// TIA Portal V17 program export: 1 tag tables, 0 data types, 2 data blocks, 8 code blocks (in call order from the OBs), 3 instance data blocks

VAR_GLOBAL   // PLC tag table "System"
   System_Byte AT %MB1 : Byte;
   FirstScan AT %M1.0 : Bool;
   DiagStatusUpdate AT %M1.1 : Bool;
   AlwaysTRUE AT %M1.2 : Bool;
   AlwaysFALSE AT %M1.3 : Bool;
   Clock_Byte AT %MB0 : Byte;
   Clock_10Hz AT %M0.0 : Bool;
   Clock_5Hz AT %M0.1 : Bool;
   "Clock_2.5Hz" AT %M0.2 : Bool;
   Clock_2Hz AT %M0.3 : Bool;
   "Clock_1.25Hz" AT %M0.4 : Bool;
   Clock_1Hz AT %M0.5 : Bool;
   "Clock_0.625Hz" AT %M0.6 : Bool;
   "Clock_0.5Hz" AT %M0.7 : Bool;
   Tag_1 AT %MD100 : DWord;
END_VAR

DATA_BLOCK "Modbus RTU buffer"   // DB11
{ S7_Optimized_Access := 'FALSE' }
VERSION : 0.1
// stored: AutoNumber false, DBAccessibleFromOPCUA true, IsOnlyStoredInLoadMemory false, IsWriteProtectedInAS false
   VAR
      "Operation data number_H" { ExternalAccessible := 'False'; ExternalVisible := 'False'; ExternalWritable := 'False'} : UInt;   // Modbus register 88
      "Operation data number_L" { ExternalAccessible := 'False'; ExternalVisible := 'False'; ExternalWritable := 'False'} : UInt;   // Modbus register 89
      "Operation type_H" { ExternalAccessible := 'False'; ExternalVisible := 'False'; ExternalWritable := 'False'} : UInt;   // Modbus register 90
      "Operation type_L" { ExternalAccessible := 'False'; ExternalVisible := 'False'; ExternalWritable := 'False'} : UInt;   // Modbus register 91
      Position_H { ExternalAccessible := 'False'; ExternalVisible := 'False'; ExternalWritable := 'False'} : UInt;   // Modbus register 92
      Position_L { ExternalAccessible := 'False'; ExternalVisible := 'False'; ExternalWritable := 'False'} : UInt;   // Modbus register 93
      Speed_H { ExternalAccessible := 'False'; ExternalVisible := 'False'; ExternalWritable := 'False'} : UInt;   // Modbus register 94
      Speed_L { ExternalAccessible := 'False'; ExternalVisible := 'False'; ExternalWritable := 'False'} : UInt;   // Modbus register 95
      "Starting_Changing rate_H" { ExternalAccessible := 'False'; ExternalVisible := 'False'; ExternalWritable := 'False'} : UInt;   // Modbus register 96
      "Starting_Changing rate_L" { ExternalAccessible := 'False'; ExternalVisible := 'False'; ExternalWritable := 'False'} : UInt;   // Modbus register 97
      "Stopping deceleration_H" { ExternalAccessible := 'False'; ExternalVisible := 'False'; ExternalWritable := 'False'} : UInt;   // Modbus register 98
      "Stopping deceleration_L" { ExternalAccessible := 'False'; ExternalVisible := 'False'; ExternalWritable := 'False'} : UInt;   // Modbus register 99
      "Operating current_H" { ExternalAccessible := 'False'; ExternalVisible := 'False'; ExternalWritable := 'False'} : UInt;   // Modbus register 100
      "Operating current_L" { ExternalAccessible := 'False'; ExternalVisible := 'False'; ExternalWritable := 'False'} : UInt;   // Modbus register 101
      "Operation trigger_H" { ExternalAccessible := 'False'; ExternalVisible := 'False'; ExternalWritable := 'False'} : UInt;   // Modbus register 102
      "Operation trigger_L" { ExternalAccessible := 'False'; ExternalVisible := 'False'; ExternalWritable := 'False'} : UInt;   // Modbus register 103
      "Forwarding destination_H" { ExternalAccessible := 'False'; ExternalVisible := 'False'; ExternalWritable := 'False'} : UInt;   // Modbus register 104
      "Forwarding destination_L" { ExternalAccessible := 'False'; ExternalVisible := 'False'; ExternalWritable := 'False'} : UInt;   // Modbus register 105
      "Alarm reset_H" { ExternalAccessible := 'False'; ExternalVisible := 'False'; ExternalWritable := 'False'} : UInt;   // Modbus register 384
      "Alarm reset_L" { ExternalAccessible := 'False'; ExternalVisible := 'False'; ExternalWritable := 'False'} : UInt;   // Modbus register 385
      "Clear Monitor alarm history_H" { ExternalAccessible := 'False'; ExternalVisible := 'False'; ExternalWritable := 'False'} : UInt;   // Modbus register 388
      "Clear Monitor alarm history_L" { ExternalAccessible := 'False'; ExternalVisible := 'False'; ExternalWritable := 'False'} : UInt;   // Modbus register 389
      "Clear comm history_H" { ExternalAccessible := 'False'; ExternalVisible := 'False'; ExternalWritable := 'False'} : UInt;   // Modbus register 392
      "Clear comm history_L" { ExternalAccessible := 'False'; ExternalVisible := 'False'; ExternalWritable := 'False'} : UInt;   // Modbus register 393
      "Monitor present alarm_H" { ExternalAccessible := 'False'; ExternalVisible := 'False'; ExternalWritable := 'False'} : UInt;   // Modbus register 128
      "Monitor present alarm_L" { ExternalAccessible := 'False'; ExternalVisible := 'False'; ExternalWritable := 'False'} : UInt;   // Modbus register 129
      "Monitor alarm history 1_H" { ExternalAccessible := 'False'; ExternalVisible := 'False'; ExternalWritable := 'False'} : UInt;   // Modbus register 130
      "Monitor alarm history 1_L" { ExternalAccessible := 'False'; ExternalVisible := 'False'; ExternalWritable := 'False'} : UInt;   // Modbus register 131
      "Monitor alarm history 2_H" { ExternalAccessible := 'False'; ExternalVisible := 'False'; ExternalWritable := 'False'} : UInt;   // Modbus register 132
      "Monitor alarm history 2_L" { ExternalAccessible := 'False'; ExternalVisible := 'False'; ExternalWritable := 'False'} : UInt;   // Modbus register 133
      "Monitor alarm history 3_H" { ExternalAccessible := 'False'; ExternalVisible := 'False'; ExternalWritable := 'False'} : UInt;   // Modbus register 134
      "Monitor alarm history 3_L" { ExternalAccessible := 'False'; ExternalVisible := 'False'; ExternalWritable := 'False'} : UInt;   // Modbus register 135
      "Monitor alarm history 4_H" { ExternalAccessible := 'False'; ExternalVisible := 'False'; ExternalWritable := 'False'} : UInt;   // Modbus register 136
      "Monitor alarm history 4_L" { ExternalAccessible := 'False'; ExternalVisible := 'False'; ExternalWritable := 'False'} : UInt;   // Modbus register 137
      "Monitor alarm history 5_H" { ExternalAccessible := 'False'; ExternalVisible := 'False'; ExternalWritable := 'False'} : UInt;   // Modbus register 138
      "Monitor alarm history 5_L" { ExternalAccessible := 'False'; ExternalVisible := 'False'; ExternalWritable := 'False'} : UInt;   // Modbus register 139
      "Monitor present communication error_H" { ExternalAccessible := 'False'; ExternalVisible := 'False'; ExternalWritable := 'False'} : UInt;   // Modbus register 172
      "Monitor present communication error_L" { ExternalAccessible := 'False'; ExternalVisible := 'False'; ExternalWritable := 'False'} : UInt;   // Modbus register 173
      "Monitor communication error history 1_H" { ExternalAccessible := 'False'; ExternalVisible := 'False'; ExternalWritable := 'False'} : UInt;   // Modbus register 174
      "Monitor communication error history 1_L" { ExternalAccessible := 'False'; ExternalVisible := 'False'; ExternalWritable := 'False'} : UInt;   // Modbus register 175
      "Monitor communication error history 2_H" { ExternalAccessible := 'False'; ExternalVisible := 'False'; ExternalWritable := 'False'} : UInt;   // Modbus register 176
      "Monitor communication error history 2_L" { ExternalAccessible := 'False'; ExternalVisible := 'False'; ExternalWritable := 'False'} : UInt;   // Modbus register 177
      "Monitor communication error history 3_H" { ExternalAccessible := 'False'; ExternalVisible := 'False'; ExternalWritable := 'False'} : UInt;   // Modbus register 178
      "Monitor communication error history 3_L" { ExternalAccessible := 'False'; ExternalVisible := 'False'; ExternalWritable := 'False'} : UInt;   // Modbus register 179
      "Monitor communication error history 4_H" { ExternalAccessible := 'False'; ExternalVisible := 'False'; ExternalWritable := 'False'} : UInt;   // Modbus register 180
      "Monitor communication error history 4_L" { ExternalAccessible := 'False'; ExternalVisible := 'False'; ExternalWritable := 'False'} : UInt;   // Modbus register 181
      "Monitor communication error history 5_H" { ExternalAccessible := 'False'; ExternalVisible := 'False'; ExternalWritable := 'False'} : UInt;   // Modbus register 182
      "Monitor communication error history 5_L" { ExternalAccessible := 'False'; ExternalVisible := 'False'; ExternalWritable := 'False'} : UInt;   // Modbus register 183
      "Monitor feedback position_H" { ExternalAccessible := 'False'; ExternalVisible := 'False'; ExternalWritable := 'False'} : UInt;   // Modbus register 204
      "Monitor feedback position_L" { ExternalAccessible := 'False'; ExternalVisible := 'False'; ExternalWritable := 'False'} : UInt;   // Modbus register 205
      "Monitor feedback speed r/min_H" { ExternalAccessible := 'False'; ExternalVisible := 'False'; ExternalWritable := 'False'} : UInt;   // Modbus register 206
      "Monitor feedback speed r/min_L" { ExternalAccessible := 'False'; ExternalVisible := 'False'; ExternalWritable := 'False'} : UInt;   // Modbus register 207
      "Monitor feedback speed Hz_H" { ExternalAccessible := 'False'; ExternalVisible := 'False'; ExternalWritable := 'False'} : UInt;   // Modbus register 208
      "Monitor feedback speed Hz_L" { ExternalAccessible := 'False'; ExternalVisible := 'False'; ExternalWritable := 'False'} : UInt;   // Modbus register 209
      "Monitor direct I/O_H" { ExternalAccessible := 'False'; ExternalVisible := 'False'; ExternalWritable := 'False'} : UInt;   // Modbus register 212
      "Monitor direct I/O_L" { ExternalAccessible := 'False'; ExternalVisible := 'False'; ExternalWritable := 'False'} : UInt;   // Modbus register 213
      "Monitor torque_H" { ExternalAccessible := 'False'; ExternalVisible := 'False'; ExternalWritable := 'False'} : UInt;   // Modbus register 214
      "Monitor torque_L" { ExternalAccessible := 'False'; ExternalVisible := 'False'; ExternalWritable := 'False'} : UInt;   // Modbus register 215
      "Monitor cumulative load_H" { ExternalAccessible := 'False'; ExternalVisible := 'False'; ExternalWritable := 'False'} : UInt;   // Modbus register 218
      "Monitor cumulative load_L" { ExternalAccessible := 'False'; ExternalVisible := 'False'; ExternalWritable := 'False'} : UInt;   // Modbus register 219
      "Monitor driver temperature_H" { ExternalAccessible := 'False'; ExternalVisible := 'False'; ExternalWritable := 'False'} : UInt;   // Modbus register 248
      "Monitor driver temperature_L" { ExternalAccessible := 'False'; ExternalVisible := 'False'; ExternalWritable := 'False'} : UInt;   // Modbus register 249
      "Monitor motor temperature_H" { ExternalAccessible := 'False'; ExternalVisible := 'False'; ExternalWritable := 'False'} : UInt;   // Modbus register 250
      "Monitor motor temperature_L" { ExternalAccessible := 'False'; ExternalVisible := 'False'; ExternalWritable := 'False'} : UInt;   // Modbus register 251
      "Monitor inverter voltage_H" { ExternalAccessible := 'False'; ExternalVisible := 'False'; ExternalWritable := 'False'} : UInt;   // Modbus register 326
      "Monitor inverter voltage_L" { ExternalAccessible := 'False'; ExternalVisible := 'False'; ExternalWritable := 'False'} : UInt;   // Modbus register 327
      "Monitor power supply voltage_H" { ExternalAccessible := 'False'; ExternalVisible := 'False'; ExternalWritable := 'False'} : UInt;   // Modbus register 328
      "Monitor power supply voltage_L" { ExternalAccessible := 'False'; ExternalVisible := 'False'; ExternalWritable := 'False'} : UInt;   // Modbus register 329
      "Monitor DIP SW_H" { ExternalAccessible := 'False'; ExternalVisible := 'False'; ExternalWritable := 'False'} : UInt;   // Modbus register 330
      "Monitor DIP SW_L" { ExternalAccessible := 'False'; ExternalVisible := 'False'; ExternalWritable := 'False'} : UInt;   // Modbus register 331
      "Monitor ROT SW0_H" { ExternalAccessible := 'False'; ExternalVisible := 'False'; ExternalWritable := 'False'} : UInt;   // Modbus register 332
      "Monitor ROT SW0_L" { ExternalAccessible := 'False'; ExternalVisible := 'False'; ExternalWritable := 'False'} : UInt;   // Modbus register 333
      "Monitor ROT SW1_H" { ExternalAccessible := 'False'; ExternalVisible := 'False'; ExternalWritable := 'False'} : UInt;   // Modbus register 334
      "Monitor ROT SW1_L" { ExternalAccessible := 'False'; ExternalVisible := 'False'; ExternalWritable := 'False'} : UInt;   // Modbus register 335
   END_VAR
BEGIN
END_DATA_BLOCK

DATA_BLOCK "Modbus RTU comm"   // DB10
{ S7_Optimized_Access := 'TRUE' }
VERSION : 0.1
// stored: AutoNumber false, DBAccessibleFromOPCUA true, IsOnlyStoredInLoadMemory false, IsRetainMemResEnabled false, IsWriteProtectedInAS false, MemoryReserve 100
   VAR
      "Setup Done" { ExternalAccessible := 'False'; ExternalVisible := 'False'; ExternalWritable := 'False'} : Bool;
      Sequencer : USInt;
      REQ { ExternalAccessible := 'False'; ExternalVisible := 'False'; ExternalWritable := 'False'} : Bool;
      BUSY : Bool;
      DONE : Bool;
      MB_ADDR { ExternalAccessible := 'False'; ExternalVisible := 'False'; ExternalWritable := 'False'} : Word;
      MODE { ExternalAccessible := 'False'; ExternalVisible := 'False'; ExternalWritable := 'False'} : USInt;
      "DATA ADDR" { ExternalAccessible := 'False'; ExternalVisible := 'False'; ExternalWritable := 'False'} : UDInt;
      DATA_LEN { ExternalAccessible := 'False'; ExternalVisible := 'False'; ExternalWritable := 'False'} : UInt;
      DATA_PTR : UInt;
   END_VAR
BEGIN
END_DATA_BLOCK

ORGANIZATION_BLOCK "Main"   // OB1, LAD, ProgramCycle
TITLE = "Main Program Sweep (Cycle)"
{ S7_Optimized_Access := 'TRUE' }
VERSION : 0.1
// stored: AutoNumber true, IsIECCheckEnabled false, SetENOAutomatically false
   VAR_INPUT
      Initial_Call : Bool;   // Initial call of this OB
      Remanence : Bool;   // =True, if remanent data are available
   END_VAR
BEGIN

REGION Network 1: Call Modbus RTU program blocks
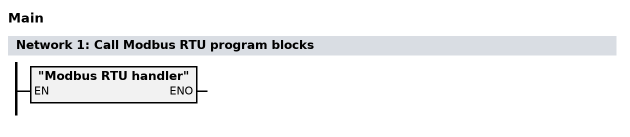
   RUNG wire#powerrail
      "Modbus RTU handler"()
   END_RUNG
   // the same network as SCL:
   "Modbus RTU handler"();
END_REGION
END_ORGANIZATION_BLOCK

FUNCTION "Modbus RTU handler" : Void   // FC10, LAD
TITLE = Modbus RTU handler
{ S7_Optimized_Access := 'TRUE' }
VERSION : 0.1
// This block updates R/W data from all the devices connected to the designated CM 1241 module.
// 
// Peripherals connected to this module:
// 
// -AZD-KD
// stored: AutoNumber false, IsIECCheckEnabled false, SetENOAutomatically false, UDAEnableTagReadback false
BEGIN

REGION Network 1: Modbus RTU module setup block
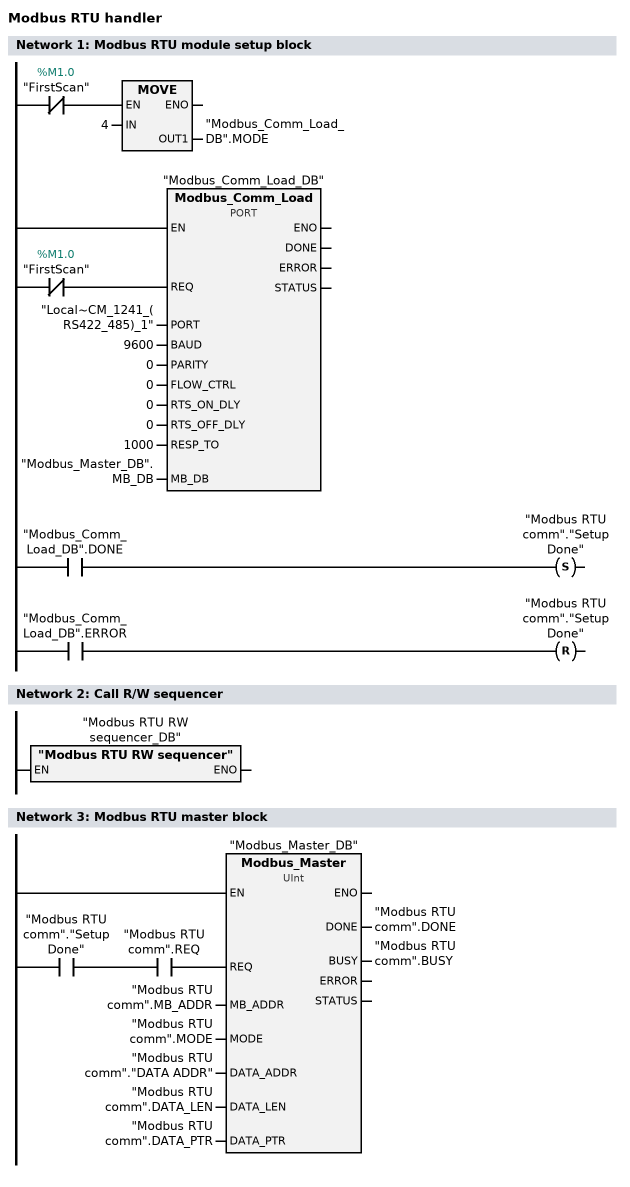
   RUNG wire#powerrail
      I_Contact( "FirstScan" )
      Move(in := 4, out1 => "Modbus_Comm_Load_DB".MODE)
   END_RUNG
   RUNG wire#powerrail
      { S7_Templates := "[card := 0, port_type := PORT, word_type := UInt, dint_type := UDInt, mbbase_type := P2P_MB_BASE]" } "Modbus_Comm_Load_DB".Modbus_Comm_Load(REQ := wire#w1, PORT := "Local~CM_1241_(RS422_485)_1", BAUD := 9600, PARITY := 0, FLOW_CTRL := 0, RTS_ON_DLY := 0, RTS_OFF_DLY := 0, RESP_TO := 1000, MB_DB := "Modbus_Master_DB".MB_DB, DONE =>, ERROR =>, STATUS =>)
   END_RUNG
   RUNG wire#powerrail
      I_Contact( "FirstScan" )
   END_RUNG wire#w1
   RUNG wire#powerrail
      Contact( "Modbus_Comm_Load_DB".DONE )
      S_Coil( "Modbus RTU comm"."Setup Done" )
   END_RUNG
   RUNG wire#powerrail
      Contact( "Modbus_Comm_Load_DB".ERROR )
      R_Coil( "Modbus RTU comm"."Setup Done" )
   END_RUNG
   // the same network as SCL:
   IF NOT "FirstScan" THEN "Modbus_Comm_Load_DB".MODE := 4; END_IF;
   "Modbus_Comm_Load_DB"(REQ := NOT "FirstScan",   // Modbus_Comm_Load
                         PORT := "Local~CM_1241_(RS422_485)_1",
                         BAUD := 9600,
                         PARITY := 0,
                         FLOW_CTRL := 0,
                         RTS_ON_DLY := 0,
                         RTS_OFF_DLY := 0,
                         RESP_TO := 1000,
                         MB_DB := "Modbus_Master_DB".MB_DB);
   IF "Modbus_Comm_Load_DB".DONE THEN "Modbus RTU comm"."Setup Done" := TRUE; END_IF;
   IF "Modbus_Comm_Load_DB".ERROR THEN "Modbus RTU comm"."Setup Done" := FALSE; END_IF;
END_REGION

REGION Network 2: Call R/W sequencer
   RUNG wire#powerrail
      "Modbus RTU RW sequencer_DB"()
   END_RUNG
   // the same network as SCL:
   "Modbus RTU RW sequencer_DB"();   // "Modbus RTU RW sequencer"
END_REGION

REGION Network 3: Modbus RTU master block
   RUNG wire#powerrail
      { S7_Templates := "[card := 0, word_type := UInt, dword_type := UDInt, byte_type := USInt, any_type := Variant]" } "Modbus_Master_DB".Modbus_Master(REQ := wire#w1, MB_ADDR := "Modbus RTU comm".MB_ADDR, MODE := "Modbus RTU comm".MODE, DATA_ADDR := "Modbus RTU comm"."DATA ADDR", DATA_LEN := "Modbus RTU comm".DATA_LEN, DATA_PTR := "Modbus RTU comm".DATA_PTR, DONE => "Modbus RTU comm".DONE, BUSY => "Modbus RTU comm".BUSY, ERROR =>, STATUS =>)
   END_RUNG
   RUNG wire#powerrail
      Contact( "Modbus RTU comm"."Setup Done" )
      Contact( "Modbus RTU comm".REQ )
   END_RUNG wire#w1
   // the same network as SCL:
   "Modbus_Master_DB"(REQ := "Modbus RTU comm"."Setup Done" AND "Modbus RTU comm".REQ,   // Modbus_Master
                      MB_ADDR := "Modbus RTU comm".MB_ADDR,
                      MODE := "Modbus RTU comm".MODE,
                      DATA_ADDR := "Modbus RTU comm"."DATA ADDR",
                      DATA_LEN := "Modbus RTU comm".DATA_LEN,
                      DATA_PTR := "Modbus RTU comm".DATA_PTR,
                      DONE => "Modbus RTU comm".DONE,
                      BUSY => "Modbus RTU comm".BUSY);
END_REGION
END_FUNCTION

FUNCTION_BLOCK "Modbus RTU RW sequencer"   // FB1, LAD
{ S7_Optimized_Access := 'TRUE' }
VERSION : 0.1
// stored: AutoNumber false, IsIECCheckEnabled false, IsRetainMemResEnabled false, MemoryReserve 100, SetENOAutomatically false, UDAEnableTagReadback false
   VAR
      "Operation data number" { S7_SetPoint := 'True'} : "Deconcatenate UDInt into two UInt";
      "Operation type" { S7_SetPoint := 'True'} : "Deconcatenate UDInt into two UInt";
      Position { S7_SetPoint := 'True'} : "Deconcatenate UDInt into two UInt";
      Speed { S7_SetPoint := 'True'} : "Deconcatenate UDInt into two UInt";
      "Starting changing rate" { S7_SetPoint := 'True'} : "Deconcatenate UDInt into two UInt";
      "Stopping deceleration" { S7_SetPoint := 'True'} : "Deconcatenate UDInt into two UInt";
      "Operating current" { S7_SetPoint := 'True'} : "Deconcatenate UDInt into two UInt";
      "Operation trigger" { S7_SetPoint := 'True'} : "Deconcatenate UDInt into two UInt";
      "Forwarding destination" { S7_SetPoint := 'True'} : "Deconcatenate UDInt into two UInt";
      "Alarm reset" { S7_SetPoint := 'True'} : "Deconcatenate UDInt into two UInt";
      "Clear alarm history" { S7_SetPoint := 'True'} : "Deconcatenate UDInt into two UInt";
      "Clear comm history" { S7_SetPoint := 'True'} : "Deconcatenate UDInt into two UInt";
      "Clear monitor alarm history" { S7_SetPoint := 'True'} : "Deconcatenate UDInt into two UInt";
      "Clear comm history_1" { S7_SetPoint := 'True'} : "Deconcatenate UDInt into two UInt";
      "Monitor present alarm" { S7_SetPoint := 'True'} : "Concatenate two UInt into one UDInt";
      "Monitor alarm history 1" { S7_SetPoint := 'True'} : "Concatenate two UInt into one UDInt";
      "Monitor alarm history 2" { S7_SetPoint := 'True'} : "Concatenate two UInt into one UDInt";
      "Monitor alarm history 3" { S7_SetPoint := 'True'} : "Concatenate two UInt into one UDInt";
      "Monitor alarm history 4" { S7_SetPoint := 'True'} : "Concatenate two UInt into one UDInt";
      "Monitor alarm history 5" { S7_SetPoint := 'True'} : "Concatenate two UInt into one UDInt";
      "Monitor present communication error" { S7_SetPoint := 'True'} : "Concatenate two UInt into one UDInt";
      "Monitor communication error history 1" { S7_SetPoint := 'True'} : "Concatenate two UInt into one UDInt";
      "Monitor communication error history 2" { S7_SetPoint := 'True'} : "Concatenate two UInt into one UDInt";
      "Monitor communication error history 3" { S7_SetPoint := 'True'} : "Concatenate two UInt into one UDInt";
      "Monitor communication error history 4" { S7_SetPoint := 'True'} : "Concatenate two UInt into one UDInt";
      "Monitor communication error history 5" { S7_SetPoint := 'True'} : "Concatenate two UInt into one UDInt";
      "Monitor feedback position" { S7_SetPoint := 'True'} : "Concatenate two UInt into one UDInt";
      "Monitor feedback speed r/min" { S7_SetPoint := 'True'} : "Concatenate two UInt into one UDInt";
      "Monitor feedback speed Hz" { S7_SetPoint := 'True'} : "Concatenate two UInt into one UDInt";
      "Monitor direct I/O" { S7_SetPoint := 'True'} : "Concatenate two UInt into one UDInt";
      "Monitor torque" { S7_SetPoint := 'True'} : "Concatenate two UInt into one UDInt";
      "Monitor cumulative load" { S7_SetPoint := 'True'} : "Concatenate two UInt into one UDInt";
      "Monitor driver temperature" { S7_SetPoint := 'True'} : "Concatenate two UInt into one UDInt";
      "Monitor motor temperature" { S7_SetPoint := 'True'} : "Concatenate two UInt into one UDInt";
      "Monitor inverter voltage" { S7_SetPoint := 'True'} : "Concatenate two UInt into one UDInt";
      "Monitor power supply voltage" { S7_SetPoint := 'True'} : "Concatenate two UInt into one UDInt";
      "Monitor DIP SW" { S7_SetPoint := 'True'} : "Concatenate two UInt into one UDInt";
      "Monitor ROT SW0" { S7_SetPoint := 'True'} : "Concatenate two UInt into one UDInt";
      "Monitor ROT SW1" { S7_SetPoint := 'True'} : "Concatenate two UInt into one UDInt";
   END_VAR
   VAR_TEMP   // added for the SCL form of the ladder/FBD networks
      _w1 : Bool;
   END_VAR
BEGIN

REGION Network 1: Deconcatenate data for writing it into modbus holding registers
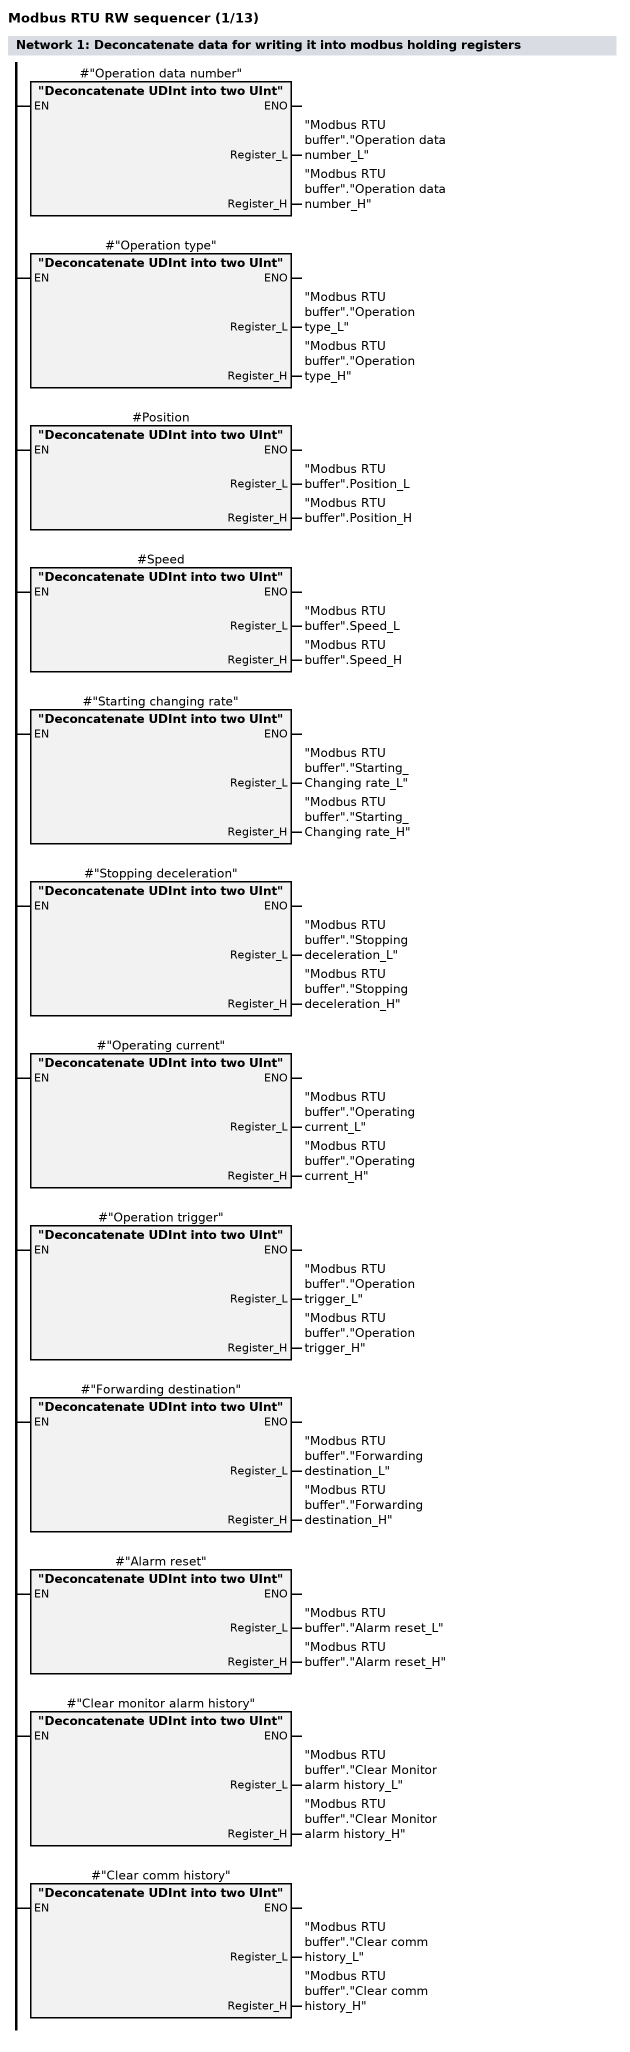
   RUNG wire#powerrail
      #"Operation data number"(Register_L => "Modbus RTU buffer"."Operation data number_L", Register_H => "Modbus RTU buffer"."Operation data number_H")
   END_RUNG
   RUNG wire#powerrail
      #"Operation type"(Register_L => "Modbus RTU buffer"."Operation type_L", Register_H => "Modbus RTU buffer"."Operation type_H")
   END_RUNG
   RUNG wire#powerrail
      #Position(Register_L => "Modbus RTU buffer".Position_L, Register_H => "Modbus RTU buffer".Position_H)
   END_RUNG
   RUNG wire#powerrail
      #Speed(Register_L => "Modbus RTU buffer".Speed_L, Register_H => "Modbus RTU buffer".Speed_H)
   END_RUNG
   RUNG wire#powerrail
      #"Starting changing rate"(Register_L => "Modbus RTU buffer"."Starting_Changing rate_L", Register_H => "Modbus RTU buffer"."Starting_Changing rate_H")
   END_RUNG
   RUNG wire#powerrail
      #"Stopping deceleration"(Register_L => "Modbus RTU buffer"."Stopping deceleration_L", Register_H => "Modbus RTU buffer"."Stopping deceleration_H")
   END_RUNG
   RUNG wire#powerrail
      #"Operating current"(Register_L => "Modbus RTU buffer"."Operating current_L", Register_H => "Modbus RTU buffer"."Operating current_H")
   END_RUNG
   RUNG wire#powerrail
      #"Operation trigger"(Register_L => "Modbus RTU buffer"."Operation trigger_L", Register_H => "Modbus RTU buffer"."Operation trigger_H")
   END_RUNG
   RUNG wire#powerrail
      #"Forwarding destination"(Register_L => "Modbus RTU buffer"."Forwarding destination_L", Register_H => "Modbus RTU buffer"."Forwarding destination_H")
   END_RUNG
   RUNG wire#powerrail
      #"Alarm reset"(Register_L => "Modbus RTU buffer"."Alarm reset_L", Register_H => "Modbus RTU buffer"."Alarm reset_H")
   END_RUNG
   RUNG wire#powerrail
      #"Clear monitor alarm history"(Register_L => "Modbus RTU buffer"."Clear Monitor alarm history_L", Register_H => "Modbus RTU buffer"."Clear Monitor alarm history_H")
   END_RUNG
   RUNG wire#powerrail
      #"Clear comm history"(Register_L => "Modbus RTU buffer"."Clear comm history_L", Register_H => "Modbus RTU buffer"."Clear comm history_H")
   END_RUNG
   // the same network as SCL:
   #"Operation data number"(Register_L => "Modbus RTU buffer"."Operation data number_L",   // "Deconcatenate UDInt into two UInt"
                           Register_H => "Modbus RTU buffer"."Operation data number_H");
   #"Operation type"(Register_L => "Modbus RTU buffer"."Operation type_L",   // "Deconcatenate UDInt into two UInt"
                     Register_H => "Modbus RTU buffer"."Operation type_H");
   #Position(Register_L => "Modbus RTU buffer".Position_L, Register_H => "Modbus RTU buffer".Position_H);   // "Deconcatenate UDInt into two UInt"
   #Speed(Register_L => "Modbus RTU buffer".Speed_L, Register_H => "Modbus RTU buffer".Speed_H);   // "Deconcatenate UDInt into two UInt"
   #"Starting changing rate"(Register_L => "Modbus RTU buffer"."Starting_Changing rate_L",   // "Deconcatenate UDInt into two UInt"
                           Register_H => "Modbus RTU buffer"."Starting_Changing rate_H");
   #"Stopping deceleration"(Register_L => "Modbus RTU buffer"."Stopping deceleration_L",   // "Deconcatenate UDInt into two UInt"
                           Register_H => "Modbus RTU buffer"."Stopping deceleration_H");
   #"Operating current"(Register_L => "Modbus RTU buffer"."Operating current_L",   // "Deconcatenate UDInt into two UInt"
                        Register_H => "Modbus RTU buffer"."Operating current_H");
   #"Operation trigger"(Register_L => "Modbus RTU buffer"."Operation trigger_L",   // "Deconcatenate UDInt into two UInt"
                        Register_H => "Modbus RTU buffer"."Operation trigger_H");
   #"Forwarding destination"(Register_L => "Modbus RTU buffer"."Forwarding destination_L",   // "Deconcatenate UDInt into two UInt"
                           Register_H => "Modbus RTU buffer"."Forwarding destination_H");
   #"Alarm reset"(Register_L => "Modbus RTU buffer"."Alarm reset_L",   // "Deconcatenate UDInt into two UInt"
                  Register_H => "Modbus RTU buffer"."Alarm reset_H");
   #"Clear monitor alarm history"(Register_L => "Modbus RTU buffer"."Clear Monitor alarm history_L",   // "Deconcatenate UDInt into two UInt"
                           Register_H => "Modbus RTU buffer"."Clear Monitor alarm history_H");
   #"Clear comm history"(Register_L => "Modbus RTU buffer"."Clear comm history_L",   // "Deconcatenate UDInt into two UInt"
                         Register_H => "Modbus RTU buffer"."Clear comm history_H");
END_REGION

REGION Network 2: Data writing/reading step 0: Write data from address 88 to address 105
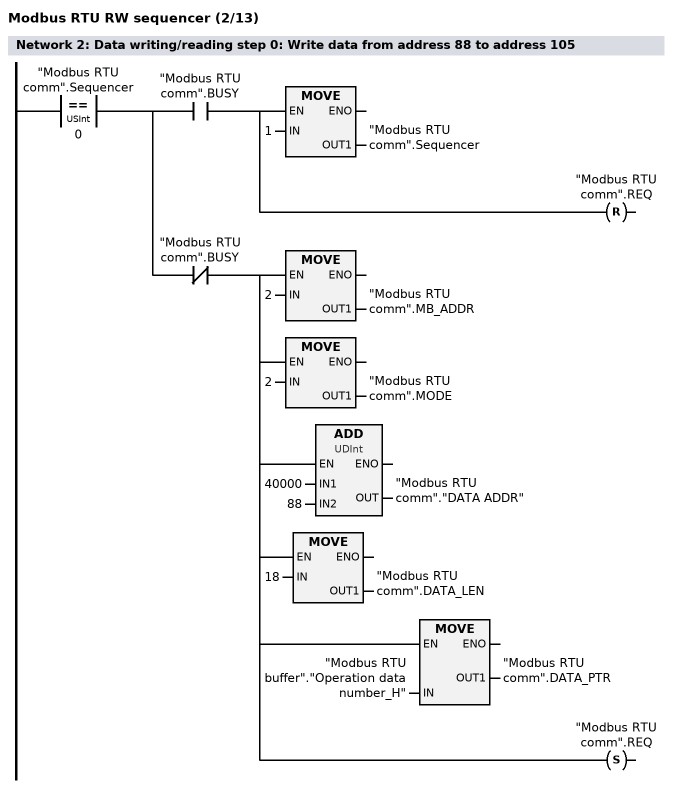
   RUNG wire#powerrail
      { S7_Templates := "SrcType := USInt" } EQ_Contact(in1 := "Modbus RTU comm".Sequencer, in2 := 0)
      wire#w1
      Contact( "Modbus RTU comm".BUSY )
      wire#w2
      Move(in := 1, out1 => "Modbus RTU comm".Sequencer)
   END_RUNG
   RUNG wire#w2
      R_Coil( "Modbus RTU comm".REQ )
   END_RUNG
   RUNG wire#w1
      I_Contact( "Modbus RTU comm".BUSY )
      wire#w3
      Move(in := 2, out1 => "Modbus RTU comm".MB_ADDR)
   END_RUNG
   RUNG wire#w3
      Move(in := 2, out1 => "Modbus RTU comm".MODE)
   END_RUNG
   RUNG wire#w3
      { S7_Templates := "SrcType := UDInt" } Add(in1 := 40000, in2 := 88, out => "Modbus RTU comm"."DATA ADDR")
   END_RUNG
   RUNG wire#w3
      Move(in := 18, out1 => "Modbus RTU comm".DATA_LEN)
   END_RUNG
   RUNG wire#w3
      Move(in := "Modbus RTU buffer"."Operation data number_H", out1 => "Modbus RTU comm".DATA_PTR)
   END_RUNG
   RUNG wire#w3
      S_Coil( "Modbus RTU comm".REQ )
   END_RUNG
   // the same network as SCL:
   #_w1 := "Modbus RTU comm".Sequencer = 0;
   IF #_w1 AND "Modbus RTU comm".BUSY THEN
       "Modbus RTU comm".Sequencer := 1;
       "Modbus RTU comm".REQ := FALSE;
   END_IF;
   IF #_w1 AND NOT "Modbus RTU comm".BUSY THEN
       "Modbus RTU comm".MB_ADDR := 2;
       "Modbus RTU comm".MODE := 2;
       "Modbus RTU comm"."DATA ADDR" := 40000 + 88;
       "Modbus RTU comm".DATA_LEN := 18;
       "Modbus RTU comm".DATA_PTR := "Modbus RTU buffer"."Operation data number_H";
       "Modbus RTU comm".REQ := TRUE;
   END_IF;
END_REGION

REGION Network 3: Data writing/reading step 1: Write data from address 384 to address 385
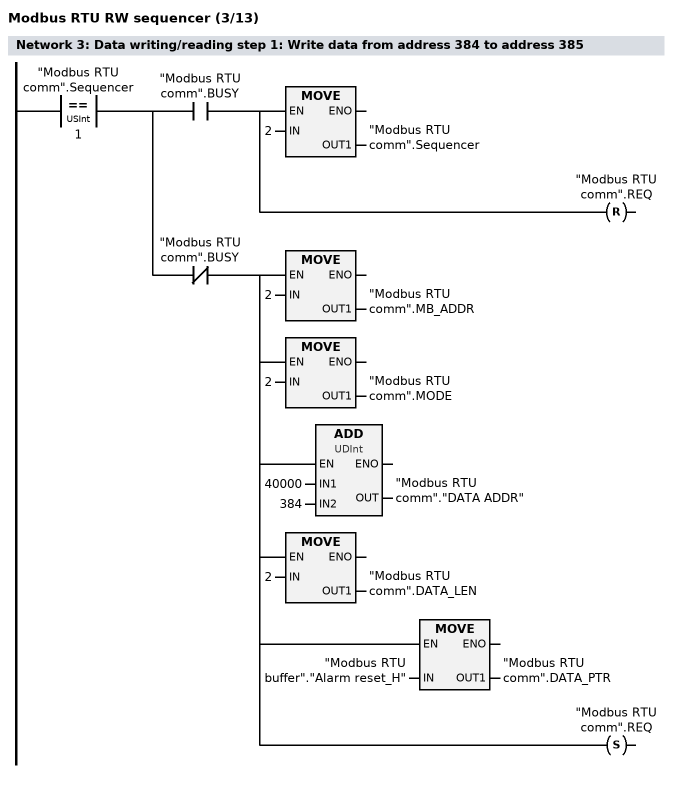
   RUNG wire#powerrail
      { S7_Templates := "SrcType := USInt" } EQ_Contact(in1 := "Modbus RTU comm".Sequencer, in2 := 1)
      wire#w1
      Contact( "Modbus RTU comm".BUSY )
      wire#w2
      Move(in := 2, out1 => "Modbus RTU comm".Sequencer)
   END_RUNG
   RUNG wire#w2
      R_Coil( "Modbus RTU comm".REQ )
   END_RUNG
   RUNG wire#w1
      I_Contact( "Modbus RTU comm".BUSY )
      wire#w3
      Move(in := 2, out1 => "Modbus RTU comm".MB_ADDR)
   END_RUNG
   RUNG wire#w3
      Move(in := 2, out1 => "Modbus RTU comm".MODE)
   END_RUNG
   RUNG wire#w3
      { S7_Templates := "SrcType := UDInt" } Add(in1 := 40000, in2 := 384, out => "Modbus RTU comm"."DATA ADDR")
   END_RUNG
   RUNG wire#w3
      Move(in := 2, out1 => "Modbus RTU comm".DATA_LEN)
   END_RUNG
   RUNG wire#w3
      Move(in := "Modbus RTU buffer"."Alarm reset_H", out1 => "Modbus RTU comm".DATA_PTR)
   END_RUNG
   RUNG wire#w3
      S_Coil( "Modbus RTU comm".REQ )
   END_RUNG
   // the same network as SCL:
   #_w1 := "Modbus RTU comm".Sequencer = 1;
   IF #_w1 AND "Modbus RTU comm".BUSY THEN
       "Modbus RTU comm".Sequencer := 2;
       "Modbus RTU comm".REQ := FALSE;
   END_IF;
   IF #_w1 AND NOT "Modbus RTU comm".BUSY THEN
       "Modbus RTU comm".MB_ADDR := 2;
       "Modbus RTU comm".MODE := 2;
       "Modbus RTU comm"."DATA ADDR" := 40000 + 384;
       "Modbus RTU comm".DATA_LEN := 2;
       "Modbus RTU comm".DATA_PTR := "Modbus RTU buffer"."Alarm reset_H";
       "Modbus RTU comm".REQ := TRUE;
   END_IF;
END_REGION

REGION Network 4: Data writing/reading step 2: Write data from address 388 to address 389
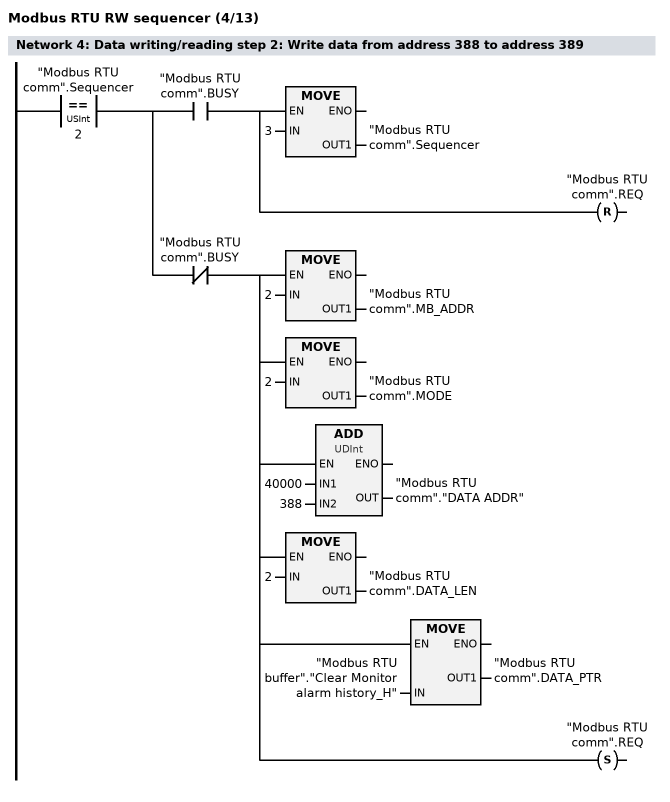
   RUNG wire#powerrail
      { S7_Templates := "SrcType := USInt" } EQ_Contact(in1 := "Modbus RTU comm".Sequencer, in2 := 2)
      wire#w1
      Contact( "Modbus RTU comm".BUSY )
      wire#w2
      Move(in := 3, out1 => "Modbus RTU comm".Sequencer)
   END_RUNG
   RUNG wire#w2
      R_Coil( "Modbus RTU comm".REQ )
   END_RUNG
   RUNG wire#w1
      I_Contact( "Modbus RTU comm".BUSY )
      wire#w3
      Move(in := 2, out1 => "Modbus RTU comm".MB_ADDR)
   END_RUNG
   RUNG wire#w3
      Move(in := 2, out1 => "Modbus RTU comm".MODE)
   END_RUNG
   RUNG wire#w3
      { S7_Templates := "SrcType := UDInt" } Add(in1 := 40000, in2 := 388, out => "Modbus RTU comm"."DATA ADDR")
   END_RUNG
   RUNG wire#w3
      Move(in := 2, out1 => "Modbus RTU comm".DATA_LEN)
   END_RUNG
   RUNG wire#w3
      Move(in := "Modbus RTU buffer"."Clear Monitor alarm history_H", out1 => "Modbus RTU comm".DATA_PTR)
   END_RUNG
   RUNG wire#w3
      S_Coil( "Modbus RTU comm".REQ )
   END_RUNG
   // the same network as SCL:
   #_w1 := "Modbus RTU comm".Sequencer = 2;
   IF #_w1 AND "Modbus RTU comm".BUSY THEN
       "Modbus RTU comm".Sequencer := 3;
       "Modbus RTU comm".REQ := FALSE;
   END_IF;
   IF #_w1 AND NOT "Modbus RTU comm".BUSY THEN
       "Modbus RTU comm".MB_ADDR := 2;
       "Modbus RTU comm".MODE := 2;
       "Modbus RTU comm"."DATA ADDR" := 40000 + 388;
       "Modbus RTU comm".DATA_LEN := 2;
       "Modbus RTU comm".DATA_PTR := "Modbus RTU buffer"."Clear Monitor alarm history_H";
       "Modbus RTU comm".REQ := TRUE;
   END_IF;
END_REGION

REGION Network 5: Data writing/reading step 3: Write data from address 392 to address 393
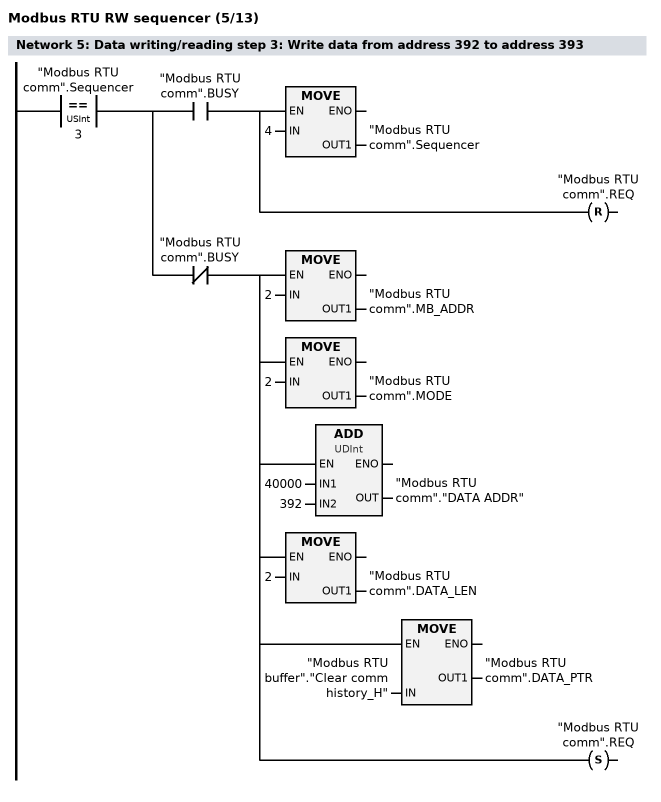
   RUNG wire#powerrail
      { S7_Templates := "SrcType := USInt" } EQ_Contact(in1 := "Modbus RTU comm".Sequencer, in2 := 3)
      wire#w1
      Contact( "Modbus RTU comm".BUSY )
      wire#w2
      Move(in := 4, out1 => "Modbus RTU comm".Sequencer)
   END_RUNG
   RUNG wire#w2
      R_Coil( "Modbus RTU comm".REQ )
   END_RUNG
   RUNG wire#w1
      I_Contact( "Modbus RTU comm".BUSY )
      wire#w3
      Move(in := 2, out1 => "Modbus RTU comm".MB_ADDR)
   END_RUNG
   RUNG wire#w3
      Move(in := 2, out1 => "Modbus RTU comm".MODE)
   END_RUNG
   RUNG wire#w3
      { S7_Templates := "SrcType := UDInt" } Add(in1 := 40000, in2 := 392, out => "Modbus RTU comm"."DATA ADDR")
   END_RUNG
   RUNG wire#w3
      Move(in := 2, out1 => "Modbus RTU comm".DATA_LEN)
   END_RUNG
   RUNG wire#w3
      Move(in := "Modbus RTU buffer"."Clear comm history_H", out1 => "Modbus RTU comm".DATA_PTR)
   END_RUNG
   RUNG wire#w3
      S_Coil( "Modbus RTU comm".REQ )
   END_RUNG
   // the same network as SCL:
   #_w1 := "Modbus RTU comm".Sequencer = 3;
   IF #_w1 AND "Modbus RTU comm".BUSY THEN
       "Modbus RTU comm".Sequencer := 4;
       "Modbus RTU comm".REQ := FALSE;
   END_IF;
   IF #_w1 AND NOT "Modbus RTU comm".BUSY THEN
       "Modbus RTU comm".MB_ADDR := 2;
       "Modbus RTU comm".MODE := 2;
       "Modbus RTU comm"."DATA ADDR" := 40000 + 392;
       "Modbus RTU comm".DATA_LEN := 2;
       "Modbus RTU comm".DATA_PTR := "Modbus RTU buffer"."Clear comm history_H";
       "Modbus RTU comm".REQ := TRUE;
   END_IF;
END_REGION

REGION Network 6: Data writing/reading step 4: Read data from address 128 to address 139
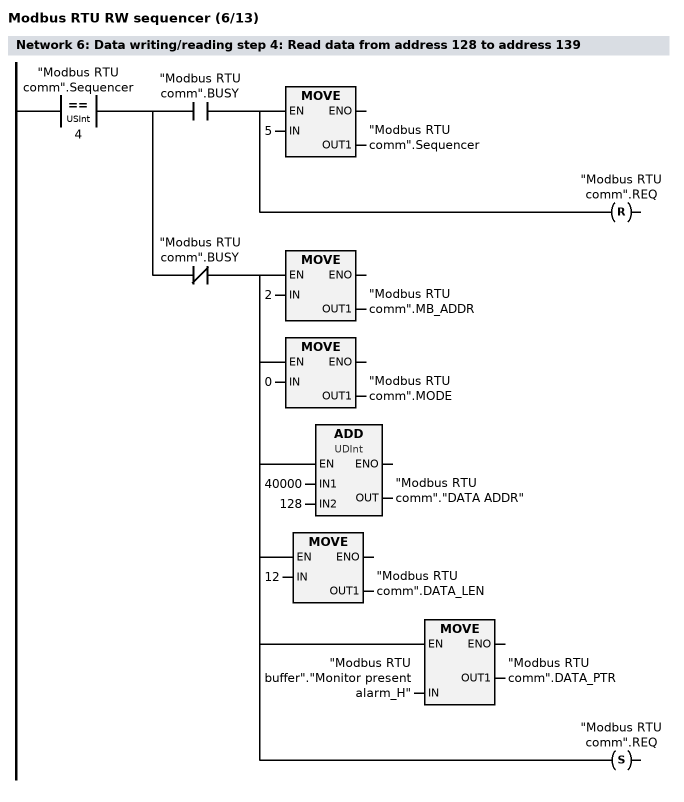
   RUNG wire#powerrail
      { S7_Templates := "SrcType := USInt" } EQ_Contact(in1 := "Modbus RTU comm".Sequencer, in2 := 4)
      wire#w1
      Contact( "Modbus RTU comm".BUSY )
      wire#w2
      Move(in := 5, out1 => "Modbus RTU comm".Sequencer)
   END_RUNG
   RUNG wire#w2
      R_Coil( "Modbus RTU comm".REQ )
   END_RUNG
   RUNG wire#w1
      I_Contact( "Modbus RTU comm".BUSY )
      wire#w3
      Move(in := 2, out1 => "Modbus RTU comm".MB_ADDR)
   END_RUNG
   RUNG wire#w3
      Move(in := 0, out1 => "Modbus RTU comm".MODE)
   END_RUNG
   RUNG wire#w3
      { S7_Templates := "SrcType := UDInt" } Add(in1 := 40000, in2 := 128, out => "Modbus RTU comm"."DATA ADDR")
   END_RUNG
   RUNG wire#w3
      Move(in := 12, out1 => "Modbus RTU comm".DATA_LEN)
   END_RUNG
   RUNG wire#w3
      Move(in := "Modbus RTU buffer"."Monitor present alarm_H", out1 => "Modbus RTU comm".DATA_PTR)
   END_RUNG
   RUNG wire#w3
      S_Coil( "Modbus RTU comm".REQ )
   END_RUNG
   // the same network as SCL:
   #_w1 := "Modbus RTU comm".Sequencer = 4;
   IF #_w1 AND "Modbus RTU comm".BUSY THEN
       "Modbus RTU comm".Sequencer := 5;
       "Modbus RTU comm".REQ := FALSE;
   END_IF;
   IF #_w1 AND NOT "Modbus RTU comm".BUSY THEN
       "Modbus RTU comm".MB_ADDR := 2;
       "Modbus RTU comm".MODE := 0;
       "Modbus RTU comm"."DATA ADDR" := 40000 + 128;
       "Modbus RTU comm".DATA_LEN := 12;
       "Modbus RTU comm".DATA_PTR := "Modbus RTU buffer"."Monitor present alarm_H";
       "Modbus RTU comm".REQ := TRUE;
   END_IF;
END_REGION

REGION Network 7: Data writing/reading step 5: Read data from address 172 to address 183
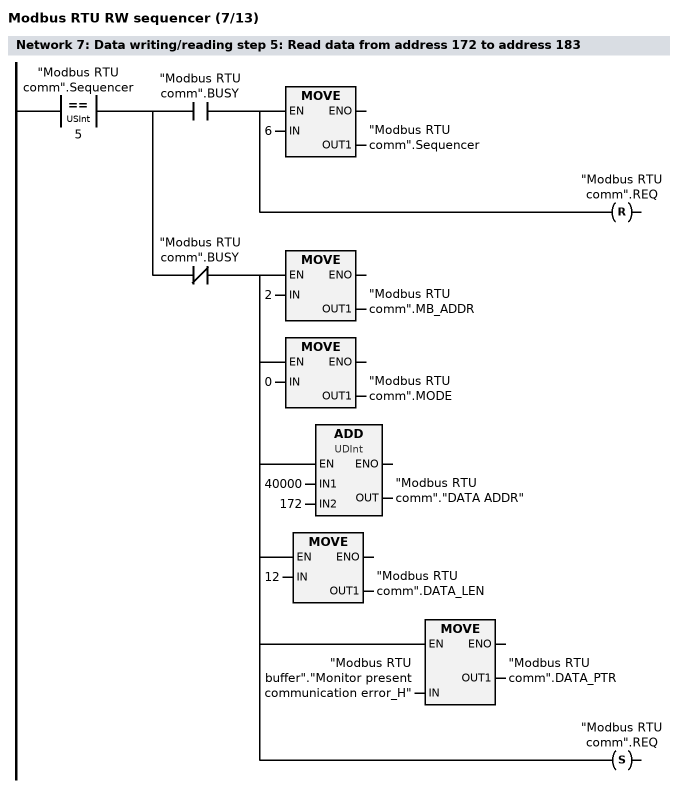
   RUNG wire#powerrail
      { S7_Templates := "SrcType := USInt" } EQ_Contact(in1 := "Modbus RTU comm".Sequencer, in2 := 5)
      wire#w1
      Contact( "Modbus RTU comm".BUSY )
      wire#w2
      Move(in := 6, out1 => "Modbus RTU comm".Sequencer)
   END_RUNG
   RUNG wire#w2
      R_Coil( "Modbus RTU comm".REQ )
   END_RUNG
   RUNG wire#w1
      I_Contact( "Modbus RTU comm".BUSY )
      wire#w3
      Move(in := 2, out1 => "Modbus RTU comm".MB_ADDR)
   END_RUNG
   RUNG wire#w3
      Move(in := 0, out1 => "Modbus RTU comm".MODE)
   END_RUNG
   RUNG wire#w3
      { S7_Templates := "SrcType := UDInt" } Add(in1 := 40000, in2 := 172, out => "Modbus RTU comm"."DATA ADDR")
   END_RUNG
   RUNG wire#w3
      Move(in := 12, out1 => "Modbus RTU comm".DATA_LEN)
   END_RUNG
   RUNG wire#w3
      Move(in := "Modbus RTU buffer"."Monitor present communication error_H", out1 => "Modbus RTU comm".DATA_PTR)
   END_RUNG
   RUNG wire#w3
      S_Coil( "Modbus RTU comm".REQ )
   END_RUNG
   // the same network as SCL:
   #_w1 := "Modbus RTU comm".Sequencer = 5;
   IF #_w1 AND "Modbus RTU comm".BUSY THEN
       "Modbus RTU comm".Sequencer := 6;
       "Modbus RTU comm".REQ := FALSE;
   END_IF;
   IF #_w1 AND NOT "Modbus RTU comm".BUSY THEN
       "Modbus RTU comm".MB_ADDR := 2;
       "Modbus RTU comm".MODE := 0;
       "Modbus RTU comm"."DATA ADDR" := 40000 + 172;
       "Modbus RTU comm".DATA_LEN := 12;
       "Modbus RTU comm".DATA_PTR := "Modbus RTU buffer"."Monitor present communication error_H";
       "Modbus RTU comm".REQ := TRUE;
   END_IF;
END_REGION

REGION Network 8: Data writing/reading step 6: Read data from address 204 to address 209
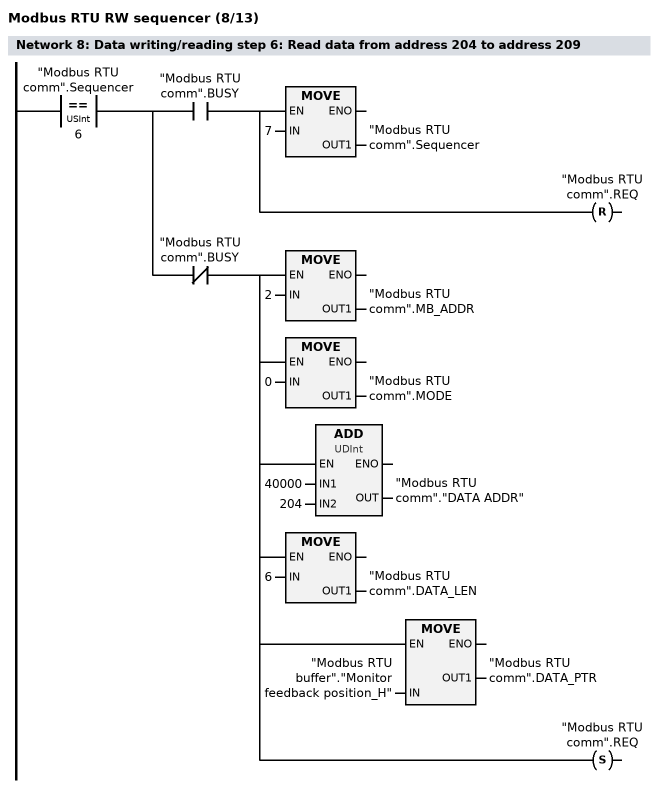
   RUNG wire#powerrail
      { S7_Templates := "SrcType := USInt" } EQ_Contact(in1 := "Modbus RTU comm".Sequencer, in2 := 6)
      wire#w1
      Contact( "Modbus RTU comm".BUSY )
      wire#w2
      Move(in := 7, out1 => "Modbus RTU comm".Sequencer)
   END_RUNG
   RUNG wire#w2
      R_Coil( "Modbus RTU comm".REQ )
   END_RUNG
   RUNG wire#w1
      I_Contact( "Modbus RTU comm".BUSY )
      wire#w3
      Move(in := 2, out1 => "Modbus RTU comm".MB_ADDR)
   END_RUNG
   RUNG wire#w3
      Move(in := 0, out1 => "Modbus RTU comm".MODE)
   END_RUNG
   RUNG wire#w3
      { S7_Templates := "SrcType := UDInt" } Add(in1 := 40000, in2 := 204, out => "Modbus RTU comm"."DATA ADDR")
   END_RUNG
   RUNG wire#w3
      Move(in := 6, out1 => "Modbus RTU comm".DATA_LEN)
   END_RUNG
   RUNG wire#w3
      Move(in := "Modbus RTU buffer"."Monitor feedback position_H", out1 => "Modbus RTU comm".DATA_PTR)
   END_RUNG
   RUNG wire#w3
      S_Coil( "Modbus RTU comm".REQ )
   END_RUNG
   // the same network as SCL:
   #_w1 := "Modbus RTU comm".Sequencer = 6;
   IF #_w1 AND "Modbus RTU comm".BUSY THEN
       "Modbus RTU comm".Sequencer := 7;
       "Modbus RTU comm".REQ := FALSE;
   END_IF;
   IF #_w1 AND NOT "Modbus RTU comm".BUSY THEN
       "Modbus RTU comm".MB_ADDR := 2;
       "Modbus RTU comm".MODE := 0;
       "Modbus RTU comm"."DATA ADDR" := 40000 + 204;
       "Modbus RTU comm".DATA_LEN := 6;
       "Modbus RTU comm".DATA_PTR := "Modbus RTU buffer"."Monitor feedback position_H";
       "Modbus RTU comm".REQ := TRUE;
   END_IF;
END_REGION

REGION Network 9: Data writing/reading step 7: Read data from address 212 to address 215
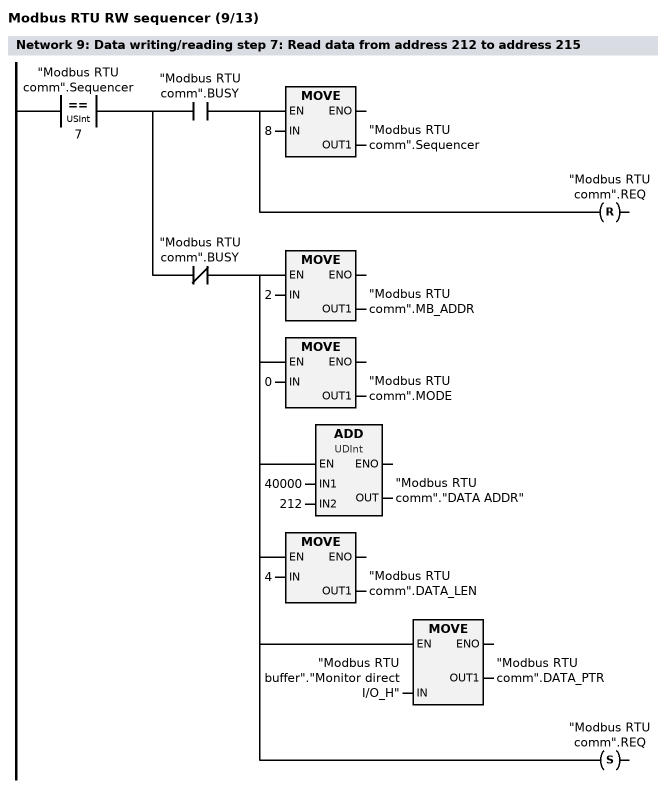
   RUNG wire#powerrail
      { S7_Templates := "SrcType := USInt" } EQ_Contact(in1 := "Modbus RTU comm".Sequencer, in2 := 7)
      wire#w1
      Contact( "Modbus RTU comm".BUSY )
      wire#w2
      Move(in := 8, out1 => "Modbus RTU comm".Sequencer)
   END_RUNG
   RUNG wire#w2
      R_Coil( "Modbus RTU comm".REQ )
   END_RUNG
   RUNG wire#w1
      I_Contact( "Modbus RTU comm".BUSY )
      wire#w3
      Move(in := 2, out1 => "Modbus RTU comm".MB_ADDR)
   END_RUNG
   RUNG wire#w3
      Move(in := 0, out1 => "Modbus RTU comm".MODE)
   END_RUNG
   RUNG wire#w3
      { S7_Templates := "SrcType := UDInt" } Add(in1 := 40000, in2 := 212, out => "Modbus RTU comm"."DATA ADDR")
   END_RUNG
   RUNG wire#w3
      Move(in := 4, out1 => "Modbus RTU comm".DATA_LEN)
   END_RUNG
   RUNG wire#w3
      Move(in := "Modbus RTU buffer"."Monitor direct I/O_H", out1 => "Modbus RTU comm".DATA_PTR)
   END_RUNG
   RUNG wire#w3
      S_Coil( "Modbus RTU comm".REQ )
   END_RUNG
   // the same network as SCL:
   #_w1 := "Modbus RTU comm".Sequencer = 7;
   IF #_w1 AND "Modbus RTU comm".BUSY THEN
       "Modbus RTU comm".Sequencer := 8;
       "Modbus RTU comm".REQ := FALSE;
   END_IF;
   IF #_w1 AND NOT "Modbus RTU comm".BUSY THEN
       "Modbus RTU comm".MB_ADDR := 2;
       "Modbus RTU comm".MODE := 0;
       "Modbus RTU comm"."DATA ADDR" := 40000 + 212;
       "Modbus RTU comm".DATA_LEN := 4;
       "Modbus RTU comm".DATA_PTR := "Modbus RTU buffer"."Monitor direct I/O_H";
       "Modbus RTU comm".REQ := TRUE;
   END_IF;
END_REGION

REGION Network 10: Data writing/reading step 8: Read data from address 218 to address 219
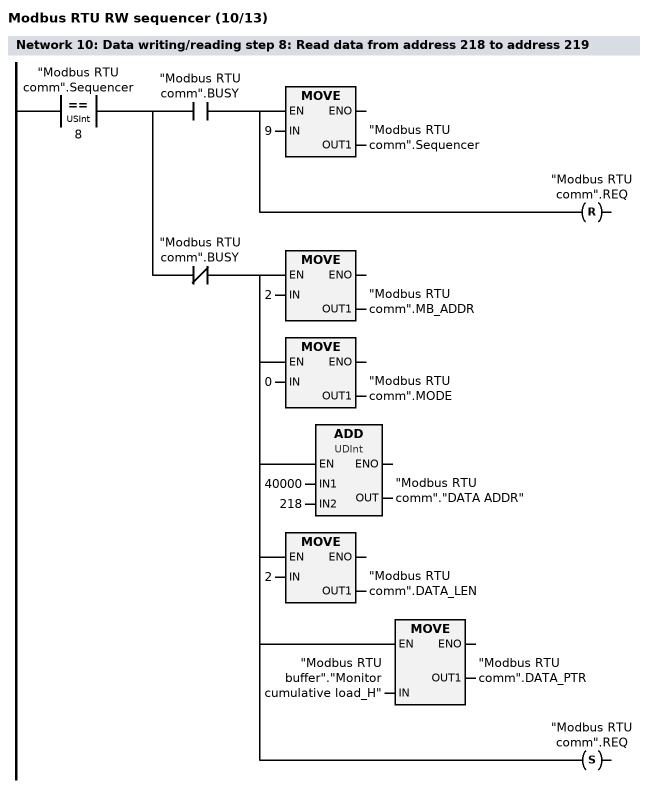
   RUNG wire#powerrail
      { S7_Templates := "SrcType := USInt" } EQ_Contact(in1 := "Modbus RTU comm".Sequencer, in2 := 8)
      wire#w1
      Contact( "Modbus RTU comm".BUSY )
      wire#w2
      Move(in := 9, out1 => "Modbus RTU comm".Sequencer)
   END_RUNG
   RUNG wire#w2
      R_Coil( "Modbus RTU comm".REQ )
   END_RUNG
   RUNG wire#w1
      I_Contact( "Modbus RTU comm".BUSY )
      wire#w3
      Move(in := 2, out1 => "Modbus RTU comm".MB_ADDR)
   END_RUNG
   RUNG wire#w3
      Move(in := 0, out1 => "Modbus RTU comm".MODE)
   END_RUNG
   RUNG wire#w3
      { S7_Templates := "SrcType := UDInt" } Add(in1 := 40000, in2 := 218, out => "Modbus RTU comm"."DATA ADDR")
   END_RUNG
   RUNG wire#w3
      Move(in := 2, out1 => "Modbus RTU comm".DATA_LEN)
   END_RUNG
   RUNG wire#w3
      Move(in := "Modbus RTU buffer"."Monitor cumulative load_H", out1 => "Modbus RTU comm".DATA_PTR)
   END_RUNG
   RUNG wire#w3
      S_Coil( "Modbus RTU comm".REQ )
   END_RUNG
   // the same network as SCL:
   #_w1 := "Modbus RTU comm".Sequencer = 8;
   IF #_w1 AND "Modbus RTU comm".BUSY THEN
       "Modbus RTU comm".Sequencer := 9;
       "Modbus RTU comm".REQ := FALSE;
   END_IF;
   IF #_w1 AND NOT "Modbus RTU comm".BUSY THEN
       "Modbus RTU comm".MB_ADDR := 2;
       "Modbus RTU comm".MODE := 0;
       "Modbus RTU comm"."DATA ADDR" := 40000 + 218;
       "Modbus RTU comm".DATA_LEN := 2;
       "Modbus RTU comm".DATA_PTR := "Modbus RTU buffer"."Monitor cumulative load_H";
       "Modbus RTU comm".REQ := TRUE;
   END_IF;
END_REGION

REGION Network 11: Data writing/reading step 9: Read data from address 248 to address 251
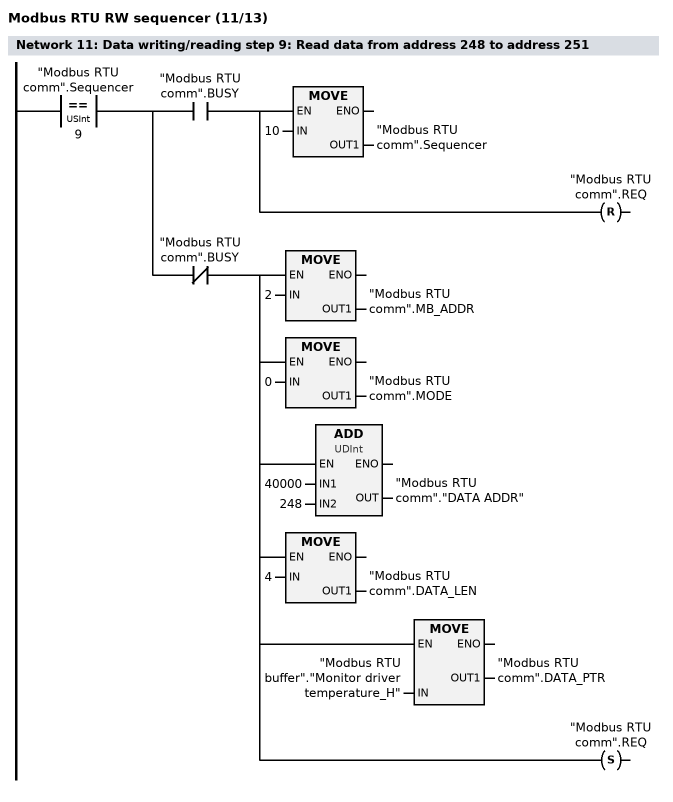
   RUNG wire#powerrail
      { S7_Templates := "SrcType := USInt" } EQ_Contact(in1 := "Modbus RTU comm".Sequencer, in2 := 9)
      wire#w1
      Contact( "Modbus RTU comm".BUSY )
      wire#w2
      Move(in := 10, out1 => "Modbus RTU comm".Sequencer)
   END_RUNG
   RUNG wire#w2
      R_Coil( "Modbus RTU comm".REQ )
   END_RUNG
   RUNG wire#w1
      I_Contact( "Modbus RTU comm".BUSY )
      wire#w3
      Move(in := 2, out1 => "Modbus RTU comm".MB_ADDR)
   END_RUNG
   RUNG wire#w3
      Move(in := 0, out1 => "Modbus RTU comm".MODE)
   END_RUNG
   RUNG wire#w3
      { S7_Templates := "SrcType := UDInt" } Add(in1 := 40000, in2 := 248, out => "Modbus RTU comm"."DATA ADDR")
   END_RUNG
   RUNG wire#w3
      Move(in := 4, out1 => "Modbus RTU comm".DATA_LEN)
   END_RUNG
   RUNG wire#w3
      Move(in := "Modbus RTU buffer"."Monitor driver temperature_H", out1 => "Modbus RTU comm".DATA_PTR)
   END_RUNG
   RUNG wire#w3
      S_Coil( "Modbus RTU comm".REQ )
   END_RUNG
   // the same network as SCL:
   #_w1 := "Modbus RTU comm".Sequencer = 9;
   IF #_w1 AND "Modbus RTU comm".BUSY THEN
       "Modbus RTU comm".Sequencer := 10;
       "Modbus RTU comm".REQ := FALSE;
   END_IF;
   IF #_w1 AND NOT "Modbus RTU comm".BUSY THEN
       "Modbus RTU comm".MB_ADDR := 2;
       "Modbus RTU comm".MODE := 0;
       "Modbus RTU comm"."DATA ADDR" := 40000 + 248;
       "Modbus RTU comm".DATA_LEN := 4;
       "Modbus RTU comm".DATA_PTR := "Modbus RTU buffer"."Monitor driver temperature_H";
       "Modbus RTU comm".REQ := TRUE;
   END_IF;
END_REGION

REGION Network 12: Data writing/reading step 10: Read data from address 326 to address 335
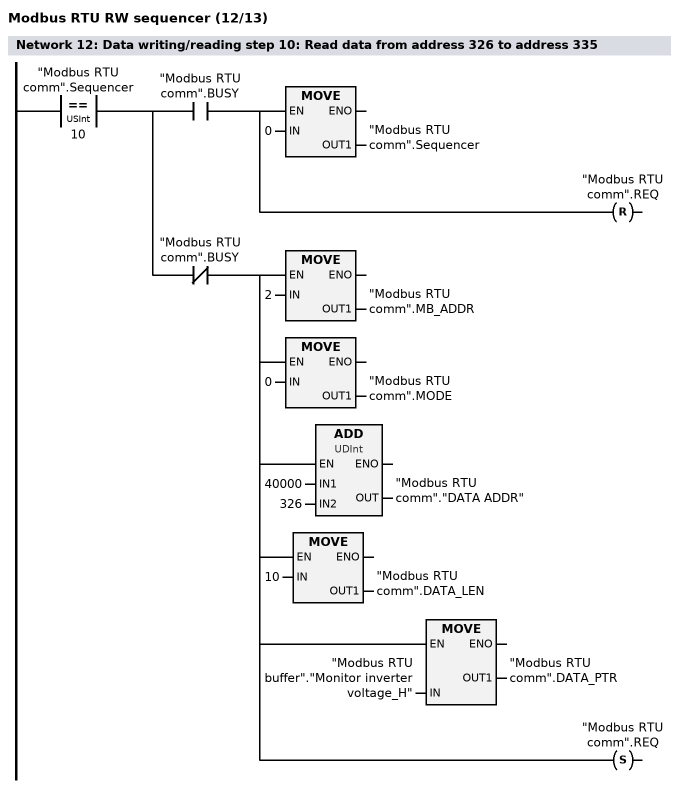
   RUNG wire#powerrail
      { S7_Templates := "SrcType := USInt" } EQ_Contact(in1 := "Modbus RTU comm".Sequencer, in2 := 10)
      wire#w1
      Contact( "Modbus RTU comm".BUSY )
      wire#w2
      Move(in := 0, out1 => "Modbus RTU comm".Sequencer)
   END_RUNG
   RUNG wire#w2
      R_Coil( "Modbus RTU comm".REQ )
   END_RUNG
   RUNG wire#w1
      I_Contact( "Modbus RTU comm".BUSY )
      wire#w3
      Move(in := 2, out1 => "Modbus RTU comm".MB_ADDR)
   END_RUNG
   RUNG wire#w3
      Move(in := 0, out1 => "Modbus RTU comm".MODE)
   END_RUNG
   RUNG wire#w3
      { S7_Templates := "SrcType := UDInt" } Add(in1 := 40000, in2 := 326, out => "Modbus RTU comm"."DATA ADDR")
   END_RUNG
   RUNG wire#w3
      Move(in := 10, out1 => "Modbus RTU comm".DATA_LEN)
   END_RUNG
   RUNG wire#w3
      Move(in := "Modbus RTU buffer"."Monitor inverter voltage_H", out1 => "Modbus RTU comm".DATA_PTR)
   END_RUNG
   RUNG wire#w3
      S_Coil( "Modbus RTU comm".REQ )
   END_RUNG
   // the same network as SCL:
   #_w1 := "Modbus RTU comm".Sequencer = 10;
   IF #_w1 AND "Modbus RTU comm".BUSY THEN
       "Modbus RTU comm".Sequencer := 0;
       "Modbus RTU comm".REQ := FALSE;
   END_IF;
   IF #_w1 AND NOT "Modbus RTU comm".BUSY THEN
       "Modbus RTU comm".MB_ADDR := 2;
       "Modbus RTU comm".MODE := 0;
       "Modbus RTU comm"."DATA ADDR" := 40000 + 326;
       "Modbus RTU comm".DATA_LEN := 10;
       "Modbus RTU comm".DATA_PTR := "Modbus RTU buffer"."Monitor inverter voltage_H";
       "Modbus RTU comm".REQ := TRUE;
   END_IF;
END_REGION

REGION Network 13: Concatenate data read from modbus holding registers into individual registers
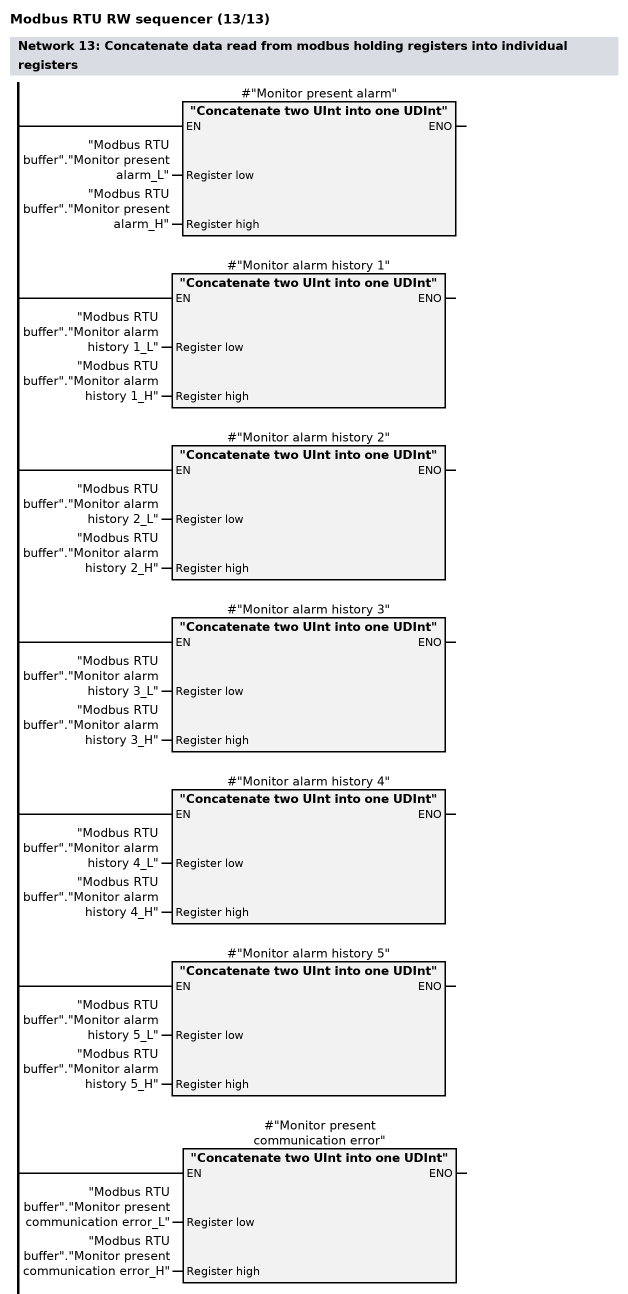
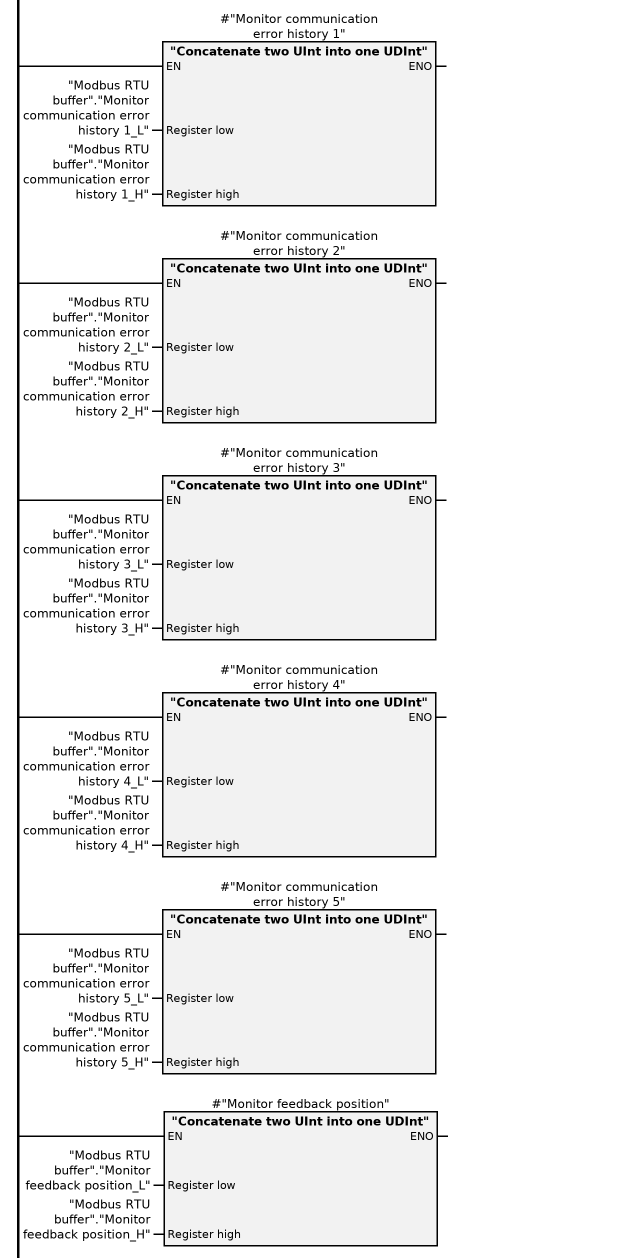
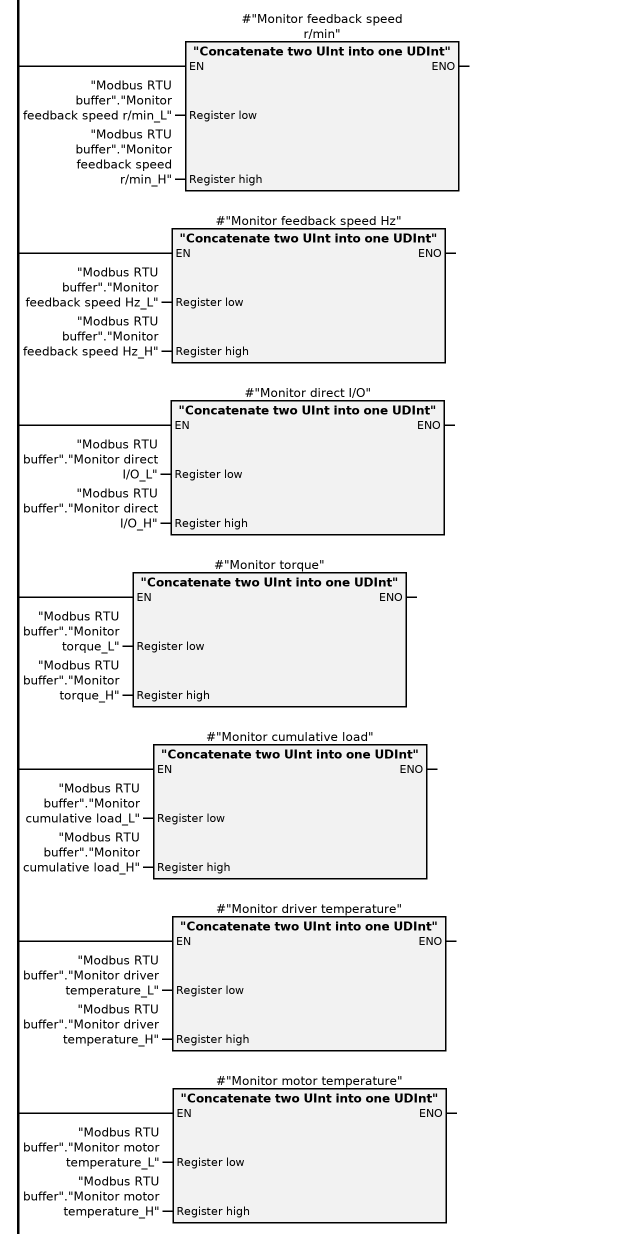
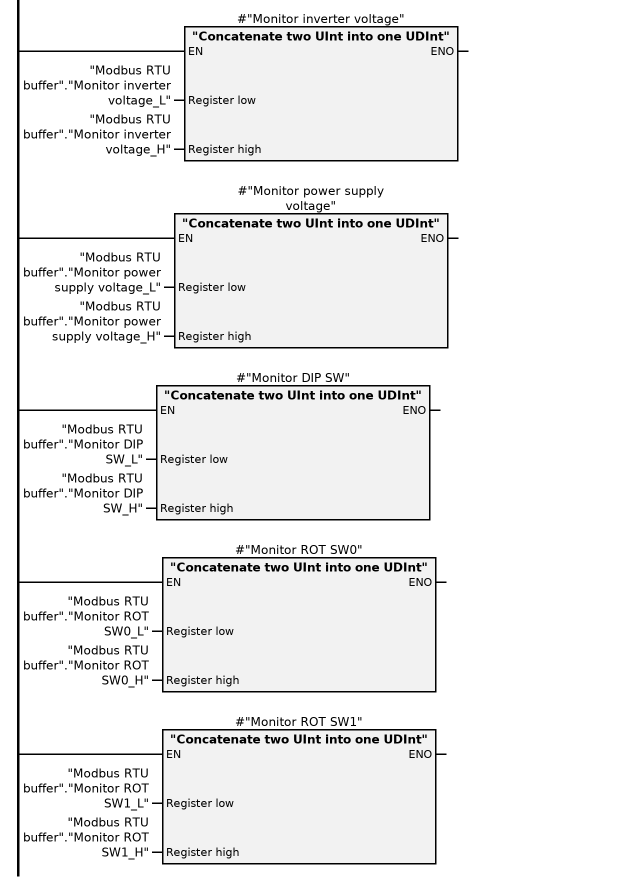
   RUNG wire#powerrail
      #"Monitor present alarm"("Register low" := "Modbus RTU buffer"."Monitor present alarm_L", "Register high" := "Modbus RTU buffer"."Monitor present alarm_H")
   END_RUNG
   RUNG wire#powerrail
      #"Monitor alarm history 1"("Register low" := "Modbus RTU buffer"."Monitor alarm history 1_L", "Register high" := "Modbus RTU buffer"."Monitor alarm history 1_H")
   END_RUNG
   RUNG wire#powerrail
      #"Monitor alarm history 2"("Register low" := "Modbus RTU buffer"."Monitor alarm history 2_L", "Register high" := "Modbus RTU buffer"."Monitor alarm history 2_H")
   END_RUNG
   RUNG wire#powerrail
      #"Monitor alarm history 3"("Register low" := "Modbus RTU buffer"."Monitor alarm history 3_L", "Register high" := "Modbus RTU buffer"."Monitor alarm history 3_H")
   END_RUNG
   RUNG wire#powerrail
      #"Monitor alarm history 4"("Register low" := "Modbus RTU buffer"."Monitor alarm history 4_L", "Register high" := "Modbus RTU buffer"."Monitor alarm history 4_H")
   END_RUNG
   RUNG wire#powerrail
      #"Monitor alarm history 5"("Register low" := "Modbus RTU buffer"."Monitor alarm history 5_L", "Register high" := "Modbus RTU buffer"."Monitor alarm history 5_H")
   END_RUNG
   RUNG wire#powerrail
      #"Monitor present communication error"("Register low" := "Modbus RTU buffer"."Monitor present communication error_L", "Register high" := "Modbus RTU buffer"."Monitor present communication error_H")
   END_RUNG
   RUNG wire#powerrail
      #"Monitor communication error history 1"("Register low" := "Modbus RTU buffer"."Monitor communication error history 1_L", "Register high" := "Modbus RTU buffer"."Monitor communication error history 1_H")
   END_RUNG
   RUNG wire#powerrail
      #"Monitor communication error history 2"("Register low" := "Modbus RTU buffer"."Monitor communication error history 2_L", "Register high" := "Modbus RTU buffer"."Monitor communication error history 2_H")
   END_RUNG
   RUNG wire#powerrail
      #"Monitor communication error history 3"("Register low" := "Modbus RTU buffer"."Monitor communication error history 3_L", "Register high" := "Modbus RTU buffer"."Monitor communication error history 3_H")
   END_RUNG
   RUNG wire#powerrail
      #"Monitor communication error history 4"("Register low" := "Modbus RTU buffer"."Monitor communication error history 4_L", "Register high" := "Modbus RTU buffer"."Monitor communication error history 4_H")
   END_RUNG
   RUNG wire#powerrail
      #"Monitor communication error history 5"("Register low" := "Modbus RTU buffer"."Monitor communication error history 5_L", "Register high" := "Modbus RTU buffer"."Monitor communication error history 5_H")
   END_RUNG
   RUNG wire#powerrail
      #"Monitor feedback position"("Register low" := "Modbus RTU buffer"."Monitor feedback position_L", "Register high" := "Modbus RTU buffer"."Monitor feedback position_H")
   END_RUNG
   RUNG wire#powerrail
      #"Monitor feedback speed r/min"("Register low" := "Modbus RTU buffer"."Monitor feedback speed r/min_L", "Register high" := "Modbus RTU buffer"."Monitor feedback speed r/min_H")
   END_RUNG
   RUNG wire#powerrail
      #"Monitor feedback speed Hz"("Register low" := "Modbus RTU buffer"."Monitor feedback speed Hz_L", "Register high" := "Modbus RTU buffer"."Monitor feedback speed Hz_H")
   END_RUNG
   RUNG wire#powerrail
      #"Monitor direct I/O"("Register low" := "Modbus RTU buffer"."Monitor direct I/O_L", "Register high" := "Modbus RTU buffer"."Monitor direct I/O_H")
   END_RUNG
   RUNG wire#powerrail
      #"Monitor torque"("Register low" := "Modbus RTU buffer"."Monitor torque_L", "Register high" := "Modbus RTU buffer"."Monitor torque_H")
   END_RUNG
   RUNG wire#powerrail
      #"Monitor cumulative load"("Register low" := "Modbus RTU buffer"."Monitor cumulative load_L", "Register high" := "Modbus RTU buffer"."Monitor cumulative load_H")
   END_RUNG
   RUNG wire#powerrail
      #"Monitor driver temperature"("Register low" := "Modbus RTU buffer"."Monitor driver temperature_L", "Register high" := "Modbus RTU buffer"."Monitor driver temperature_H")
   END_RUNG
   RUNG wire#powerrail
      #"Monitor motor temperature"("Register low" := "Modbus RTU buffer"."Monitor motor temperature_L", "Register high" := "Modbus RTU buffer"."Monitor motor temperature_H")
   END_RUNG
   RUNG wire#powerrail
      #"Monitor inverter voltage"("Register low" := "Modbus RTU buffer"."Monitor inverter voltage_L", "Register high" := "Modbus RTU buffer"."Monitor inverter voltage_H")
   END_RUNG
   RUNG wire#powerrail
      #"Monitor power supply voltage"("Register low" := "Modbus RTU buffer"."Monitor power supply voltage_L", "Register high" := "Modbus RTU buffer"."Monitor power supply voltage_H")
   END_RUNG
   RUNG wire#powerrail
      #"Monitor DIP SW"("Register low" := "Modbus RTU buffer"."Monitor DIP SW_L", "Register high" := "Modbus RTU buffer"."Monitor DIP SW_H")
   END_RUNG
   RUNG wire#powerrail
      #"Monitor ROT SW0"("Register low" := "Modbus RTU buffer"."Monitor ROT SW0_L", "Register high" := "Modbus RTU buffer"."Monitor ROT SW0_H")
   END_RUNG
   RUNG wire#powerrail
      #"Monitor ROT SW1"("Register low" := "Modbus RTU buffer"."Monitor ROT SW1_L", "Register high" := "Modbus RTU buffer"."Monitor ROT SW1_H")
   END_RUNG
   // the same network as SCL:
   #"Monitor present alarm"("Register low" := "Modbus RTU buffer"."Monitor present alarm_L",   // "Concatenate two UInt into one UDInt"
                           "Register high" := "Modbus RTU buffer"."Monitor present alarm_H");
   #"Monitor alarm history 1"("Register low" := "Modbus RTU buffer"."Monitor alarm history 1_L",   // "Concatenate two UInt into one UDInt"
                           "Register high" := "Modbus RTU buffer"."Monitor alarm history 1_H");
   #"Monitor alarm history 2"("Register low" := "Modbus RTU buffer"."Monitor alarm history 2_L",   // "Concatenate two UInt into one UDInt"
                           "Register high" := "Modbus RTU buffer"."Monitor alarm history 2_H");
   #"Monitor alarm history 3"("Register low" := "Modbus RTU buffer"."Monitor alarm history 3_L",   // "Concatenate two UInt into one UDInt"
                           "Register high" := "Modbus RTU buffer"."Monitor alarm history 3_H");
   #"Monitor alarm history 4"("Register low" := "Modbus RTU buffer"."Monitor alarm history 4_L",   // "Concatenate two UInt into one UDInt"
                           "Register high" := "Modbus RTU buffer"."Monitor alarm history 4_H");
   #"Monitor alarm history 5"("Register low" := "Modbus RTU buffer"."Monitor alarm history 5_L",   // "Concatenate two UInt into one UDInt"
                           "Register high" := "Modbus RTU buffer"."Monitor alarm history 5_H");
   #"Monitor present communication error"("Register low" := "Modbus RTU buffer"."Monitor present communication error_L",   // "Concatenate two UInt into one UDInt"
                           "Register high" := "Modbus RTU buffer"."Monitor present communication error_H");
   #"Monitor communication error history 1"("Register low" := "Modbus RTU buffer"."Monitor communication error history 1_L",   // "Concatenate two UInt into one UDInt"
                           "Register high" := "Modbus RTU buffer"."Monitor communication error history 1_H");
   #"Monitor communication error history 2"("Register low" := "Modbus RTU buffer"."Monitor communication error history 2_L",   // "Concatenate two UInt into one UDInt"
                           "Register high" := "Modbus RTU buffer"."Monitor communication error history 2_H");
   #"Monitor communication error history 3"("Register low" := "Modbus RTU buffer"."Monitor communication error history 3_L",   // "Concatenate two UInt into one UDInt"
                           "Register high" := "Modbus RTU buffer"."Monitor communication error history 3_H");
   #"Monitor communication error history 4"("Register low" := "Modbus RTU buffer"."Monitor communication error history 4_L",   // "Concatenate two UInt into one UDInt"
                           "Register high" := "Modbus RTU buffer"."Monitor communication error history 4_H");
   #"Monitor communication error history 5"("Register low" := "Modbus RTU buffer"."Monitor communication error history 5_L",   // "Concatenate two UInt into one UDInt"
                           "Register high" := "Modbus RTU buffer"."Monitor communication error history 5_H");
   #"Monitor feedback position"("Register low" := "Modbus RTU buffer"."Monitor feedback position_L",   // "Concatenate two UInt into one UDInt"
                           "Register high" := "Modbus RTU buffer"."Monitor feedback position_H");
   #"Monitor feedback speed r/min"("Register low" := "Modbus RTU buffer"."Monitor feedback speed r/min_L",   // "Concatenate two UInt into one UDInt"
                           "Register high" := "Modbus RTU buffer"."Monitor feedback speed r/min_H");
   #"Monitor feedback speed Hz"("Register low" := "Modbus RTU buffer"."Monitor feedback speed Hz_L",   // "Concatenate two UInt into one UDInt"
                           "Register high" := "Modbus RTU buffer"."Monitor feedback speed Hz_H");
   #"Monitor direct I/O"("Register low" := "Modbus RTU buffer"."Monitor direct I/O_L",   // "Concatenate two UInt into one UDInt"
                         "Register high" := "Modbus RTU buffer"."Monitor direct I/O_H");
   #"Monitor torque"("Register low" := "Modbus RTU buffer"."Monitor torque_L",   // "Concatenate two UInt into one UDInt"
                     "Register high" := "Modbus RTU buffer"."Monitor torque_H");
   #"Monitor cumulative load"("Register low" := "Modbus RTU buffer"."Monitor cumulative load_L",   // "Concatenate two UInt into one UDInt"
                           "Register high" := "Modbus RTU buffer"."Monitor cumulative load_H");
   #"Monitor driver temperature"("Register low" := "Modbus RTU buffer"."Monitor driver temperature_L",   // "Concatenate two UInt into one UDInt"
                           "Register high" := "Modbus RTU buffer"."Monitor driver temperature_H");
   #"Monitor motor temperature"("Register low" := "Modbus RTU buffer"."Monitor motor temperature_L",   // "Concatenate two UInt into one UDInt"
                           "Register high" := "Modbus RTU buffer"."Monitor motor temperature_H");
   #"Monitor inverter voltage"("Register low" := "Modbus RTU buffer"."Monitor inverter voltage_L",   // "Concatenate two UInt into one UDInt"
                           "Register high" := "Modbus RTU buffer"."Monitor inverter voltage_H");
   #"Monitor power supply voltage"("Register low" := "Modbus RTU buffer"."Monitor power supply voltage_L",   // "Concatenate two UInt into one UDInt"
                           "Register high" := "Modbus RTU buffer"."Monitor power supply voltage_H");
   #"Monitor DIP SW"("Register low" := "Modbus RTU buffer"."Monitor DIP SW_L",   // "Concatenate two UInt into one UDInt"
                     "Register high" := "Modbus RTU buffer"."Monitor DIP SW_H");
   #"Monitor ROT SW0"("Register low" := "Modbus RTU buffer"."Monitor ROT SW0_L",   // "Concatenate two UInt into one UDInt"
                      "Register high" := "Modbus RTU buffer"."Monitor ROT SW0_H");
   #"Monitor ROT SW1"("Register low" := "Modbus RTU buffer"."Monitor ROT SW1_L",   // "Concatenate two UInt into one UDInt"
                      "Register high" := "Modbus RTU buffer"."Monitor ROT SW1_H");
END_REGION
END_FUNCTION_BLOCK

FUNCTION_BLOCK "Deconcatenate UDInt into two UInt"
{ S7_Optimized_Access := 'TRUE' }
VERSION : 0.1
   VAR_OUTPUT 
      Register_L : UInt;
      Register_H { ExternalAccessible := 'False'; ExternalVisible := 'False'; ExternalWritable := 'False'} : UInt;
   END_VAR

   VAR 
      Register : UDInt;
   END_VAR

   VAR_TEMP 
      Temp : UDInt;
   END_VAR


BEGIN
	#Register_L := UDINT_TO_UINT(#Register);
	#Temp := SHR_UDINT(IN := #Temp, N := 16);
	#Register_H := UDINT_TO_UINT(#Temp); 
END_FUNCTION_BLOCK

FUNCTION_BLOCK "Concatenate two UInt into one UDInt"
{ S7_Optimized_Access := 'TRUE' }
VERSION : 0.1
   VAR_INPUT 
      "Register low" { ExternalAccessible := 'False'; ExternalVisible := 'False'; ExternalWritable := 'False'} : UInt;
      "Register high" { ExternalAccessible := 'False'; ExternalVisible := 'False'; ExternalWritable := 'False'} : UInt;
   END_VAR

   VAR 
      Register { ExternalAccessible := 'False'; ExternalVisible := 'False'; ExternalWritable := 'False'} : UDInt;
   END_VAR

   VAR_TEMP 
      Temp : UDInt;
   END_VAR


BEGIN
	#Temp := UINT_TO_UDINT(#"Register low");
	#Register := #Temp;
	#Temp := UINT_TO_UDINT(#"Register high");
	#Register:= #Register OR #Temp;
END_FUNCTION_BLOCK

ORGANIZATION_BLOCK "Startup"   // OB100, LAD, Startup
TITLE = "Complete Restart"
{ S7_Optimized_Access := 'TRUE' }
VERSION : 0.1
// stored: AutoNumber true, IsIECCheckEnabled false, SetENOAutomatically false
   VAR_INPUT
      LostRetentive : Bool;   // True if retentive data are lost
      LostRTC : Bool;   // True if date and time are lost
   END_VAR
BEGIN

REGION Network 1: Stepper initial values
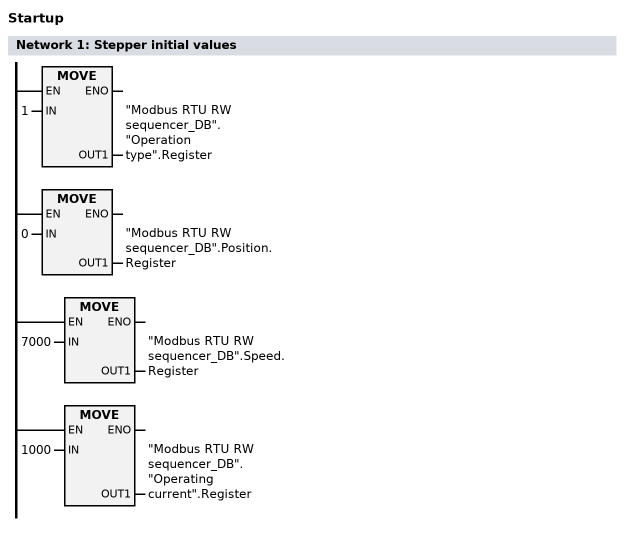
   RUNG wire#powerrail
      Move(in := 1, out1 => "Modbus RTU RW sequencer_DB"."Operation type".Register)
   END_RUNG
   RUNG wire#powerrail
      Move(in := 0, out1 => "Modbus RTU RW sequencer_DB".Position.Register)
   END_RUNG
   RUNG wire#powerrail
      Move(in := 7000, out1 => "Modbus RTU RW sequencer_DB".Speed.Register)
   END_RUNG
   RUNG wire#powerrail
      Move(in := 1000, out1 => "Modbus RTU RW sequencer_DB"."Operating current".Register)
   END_RUNG
   // the same network as SCL:
   "Modbus RTU RW sequencer_DB"."Operation type".Register := 1;
   "Modbus RTU RW sequencer_DB".Position.Register := 0;
   "Modbus RTU RW sequencer_DB".Speed.Register := 7000;
   "Modbus RTU RW sequencer_DB"."Operating current".Register := 1000;
END_REGION
END_ORGANIZATION_BLOCK

FUNCTION "Automatic sequence 1" : Void   // FC101, LAD
{ S7_Optimized_Access := 'TRUE' }
VERSION : 0.1
// stored: AutoNumber false, IsIECCheckEnabled false, SetENOAutomatically false, UDAEnableTagReadback false
BEGIN
END_FUNCTION

FUNCTION "Valves" : Void   // FC1050, FBD
{ S7_Optimized_Access := 'TRUE' }
VERSION : 0.1
// stored: AutoNumber false, IsIECCheckEnabled false, SetENOAutomatically false, UDAEnableTagReadback false
   VAR_INPUT
      "Motion enable" : Bool;
      Trigger : Bool;
      "Auto mode" : Bool;
      "Manual mode" : Bool;
      "HMI S12" : Bool;
      "HMI S14" : Bool;
      "S12 sensors" : Bool;
      "S14 sensors" : Bool;
      "S12 motion time" : Time;
      "S14 motion time" : Time;
   END_VAR
   VAR_OUTPUT
      S12 : Bool;
      S14 : Bool;
      "Alarm motion code" : USInt;
   END_VAR
   VAR_IN_OUT
      "S12 motion timer" : TON_TIME;
      "S14 motion timer" : TON_TIME;
   END_VAR
   VAR_TEMP
      "temp S12" : Bool;
      "temp S14" : Bool;
      "temp S12 motion fault" : Bool;
      "temp S14 motion fault" : Bool;
   END_VAR
   VAR_TEMP   // added for the SCL form of the ladder/FBD networks
      _w1 : Bool;
   END_VAR
BEGIN

REGION Network 1: Control logic
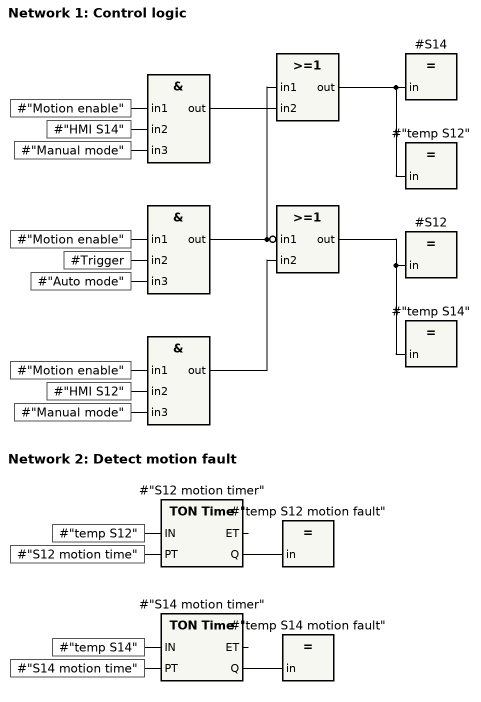
   #_w1 := #"Motion enable" AND #Trigger AND #"Auto mode";
   #S14 := #_w1 OR (#"Motion enable" AND #"HMI S14" AND #"Manual mode");
   #"temp S12" := #S14;
   #S12 := NOT #_w1 OR (#"Motion enable" AND #"HMI S12" AND #"Manual mode");
   #"temp S14" := #S12;
END_REGION

REGION Network 2: Detect motion fault
   #"S12 motion timer"(IN := #"temp S12", PT := #"S12 motion time");   // TON
   #"temp S12 motion fault" := #"S12 motion timer".Q;
   #"S14 motion timer"(IN := #"temp S14", PT := #"S14 motion time");   // TON
   #"temp S14 motion fault" := #"S14 motion timer".Q;
END_REGION

REGION Network 3: Motion alarms
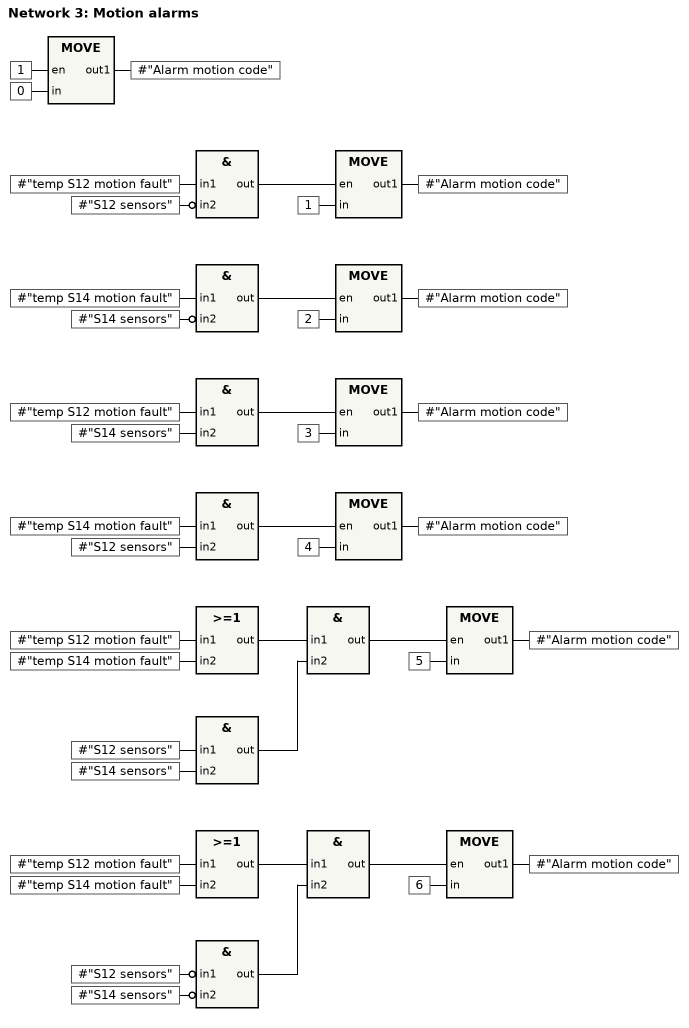
   IF 1 THEN #"Alarm motion code" := 0; END_IF;
   IF #"temp S12 motion fault" AND NOT #"S12 sensors" THEN #"Alarm motion code" := 1; END_IF;
   IF #"temp S14 motion fault" AND NOT #"S14 sensors" THEN #"Alarm motion code" := 2; END_IF;
   IF #"temp S12 motion fault" AND #"S14 sensors" THEN #"Alarm motion code" := 3; END_IF;
   IF #"temp S14 motion fault" AND #"S12 sensors" THEN #"Alarm motion code" := 4; END_IF;
   IF (#"temp S12 motion fault" OR #"temp S14 motion fault") AND #"S12 sensors" AND #"S14 sensors" THEN
       #"Alarm motion code" := 5;
   END_IF;
   IF (#"temp S12 motion fault" OR #"temp S14 motion fault") AND NOT #"S12 sensors" AND NOT #"S14 sensors" THEN
       #"Alarm motion code" := 6;
   END_IF;
END_REGION
END_FUNCTION

DATA_BLOCK "Modbus RTU RW sequencer_DB"   // DB5002
VERSION : 0.1
// stored: AutoNumber false, DBAccessibleFromOPCUA true, InstanceOfName Modbus RTU RW sequencer, InstanceOfType FB
"Modbus RTU RW sequencer"
BEGIN
END_DATA_BLOCK

DATA_BLOCK "Modbus_Comm_Load_DB"   // DB5000
// stored: AutoNumber false, DBAccessibleFromOPCUA true, InstanceOfName Modbus_Comm_Load, OfSystemLibElement Modbus_Comm_Load, OfSystemLibVersion 3.1
"Modbus_Comm_Load"
   // VAR_INPUT
   //    REQ : Bool;
   //    PORT : PORT;
   //    BAUD : UDInt;
   //    PARITY : UInt;
   //    FLOW_CTRL : UInt;
   //    RTS_ON_DLY : UInt;
   //    RTS_OFF_DLY : UInt;
   //    RESP_TO : UInt;
   // END_VAR
   // VAR_OUTPUT
   //    DONE : Bool;
   //    ERROR : Bool;
   //    STATUS : Word;
   // END_VAR
   // VAR_IN_OUT
   //    MB_DB : P2P_MB_BASE;
   // END_VAR
   // VAR
   //    ICHAR_GAP : Word;
   //    RETRIES : Word;
   //    MODE : USInt;
   //    LINE_PRE : USInt;
   //    BRK_DET : USInt;
   //    EN_DIAG_ALARM : Bool;
   //    STOP_BITS : USInt;
   //    EN_SUPPLY_VOLT : Bool;
   //    b_e_REQ : Bool;
   //    y_state : SInt;
   //    Send_Config { S7_SetPoint := 'True'} : Send_Config;
   //    Receive_Config { S7_SetPoint := 'True'} : Receive_Config;
   //    Receive_Conditions { S7_SetPoint := 'True'} : Receive_Conditions;
   //    WRREC { S7_SetPoint := 'True'} : WRREC;
   //    RDREC { S7_SetPoint := 'True'} : RDREC;
   //    port_w_record { ExternalVisible := 'False'; S7_SetPoint := 'True'} : P2P_MB_PortData;
   //    err_record { ExternalVisible := 'False'; S7_SetPoint := 'True'} : P2P_RdEstat;
   //    ftrs_w_record { ExternalVisible := 'False'; S7_SetPoint := 'True'} : P2P_FeaturesData;
   //    wlen : UInt;
   // END_VAR
BEGIN
END_DATA_BLOCK

DATA_BLOCK "Modbus_Master_DB"   // DB5001
// stored: AutoNumber false, DBAccessibleFromOPCUA true, InstanceOfName Modbus_Master, OfSystemLibElement Modbus_Master, OfSystemLibVersion 3.3
"Modbus_Master"
   // VAR_INPUT
   //    REQ : Bool;
   //    MB_ADDR : UInt;
   //    MODE : USInt;
   //    DATA_ADDR : UDInt;
   //    DATA_LEN : UInt;
   // END_VAR
   // VAR_OUTPUT
   //    DONE : Bool;
   //    BUSY : Bool;
   //    ERROR : Bool;
   //    STATUS : Word;
   // END_VAR
   // VAR_IN_OUT
   //    DATA_PTR : Variant;
   // END_VAR
   // VAR
   //    MB_State : SInt;
   //    Blocked_Proc_Timeout : Real;
   //    Extended_Addressing : Bool;
   //    Compatibility_Mode : Bool;
   //    MB_DB { S7_SetPoint := 'True'} : P2P_MB_BASE;
   //    Send_P2P { S7_SetPoint := 'True'} : Send_P2P;
   //    Receive_P2P { S7_SetPoint := 'True'} : Receive_P2P;
   //    Receive_Reset { S7_SetPoint := 'True'} : Receive_Reset;
   //    S_PORT : Word;
   //    S_RESP_TO : Word;
   //    S_ICHAR_GAP : Word;
   //    S_RETRIES : Word;
   //    S_MB_ADDR : UInt;
   //    S_MODE : USInt;
   //    S_DATA_ADDR : UDInt;
   //    S_DATA_LEN : UInt;
   //    w_retries : Word;
   //    y_SlaveAddrHi : Byte;
   //    y_SlaveAddrLo : Byte;
   //    StartAddress : Word;
   //    Value : Word;
   //    y_FCode : Byte;
   //    INTERNAL_CDATA : Array[1..257] of Byte;
   //    mb_timer { S7_SetPoint := 'True'} : TON_TIME;
   //    TimeElapsed : Bool;
   // END_VAR
BEGIN
END_DATA_BLOCK
